(* CODESYS project RPI 3b stand it.project

Project tree, tasks and I/O mapping:
  Device : CODESYS Control for Raspberry Pi SL, 3S - Smart Software Solutions GmbH, version 3.5.12.30
    application Application
      libraries: Standard, * (System); VisuDialogs, * (System)
      task MainTask (cyclic, interval 4 ms, priority 1) calls PLC_PRG
      task TrendRecordingTask (cyclic, interval 100 ms, priority 0) calls VisuTrendStorageAccess.GlobalInstances.g_TrendRecordingManager.CyclicCall
      task VISU_TASK (cyclic, interval 50 ms, priority 0) calls VisuElems.Visu_Prg
      global variables GVL
      visualisation Operator_panel
      Trend Recording Manager
        Visualization_Trend3
        Visualization_Trend2
        Operator_panel_Trend3
      Symbols
      program PLC_PRG [FBD]
      visualisation Experiment_settings
      visualisation Login
      function AfterLogin [ST]
      visualisation Settings_WGR
      visualisation Visualization
      visualisation Well_not_killed_10min
      program MySQL [ST]
      program MySQL_VISU [CFC]
      visualisation MySQL_visu
    SPI
    I²C
    SoftMotion General Axis Pool
    Modbus_COM_1 : Modbus COM, 3S - Smart Software Solutions GmbH, version 3.5.11.20
        settings: DataBits = 8; StopBits = 1; ComPort = 1
      Modbus_Master_COM_Port : Modbus Master, COM Port, 3S - Smart Software Solutions GmbH, version 3.5.12.0
          settings: Transmission = 'RTU'; ResponseTimeout = 1000; TimeBetweenFrames = 10; Auto-restart communication = TRUE
        SI30_Water_In_Add4 : Modbus Slave, COM Port, 3S - Smart Software Solutions GmbH, version 3.5.10.30
            settings: SlaveAddress = 4; ResponseTimeout = 1000; UseExtendedFunctionCodes = TRUE; Channel 2.Function Code = 5; Channel 2.Read Offset = 0; Channel 2.Read Length = 0; Channel 2.Write Offset = 16#0002; Channel 2.Write Length = 1; Channel 2.Cycle Time = 100; Channel 1.Function Code = 4; Channel 1.Read Offset = 16#0000; Channel 1.Read Length = 2; Channel 1.Write Offset = 0; Channel 1.Write Length = 0; Channel 1.Cycle Time = 100
            output Application.PLC_PRG.Reset_SI30_Waterflow_in : ARRAY[0..0] OF BYTE  // Channel 2
            input  Application.PLC_PRG.MB_Counter1_water_in : WORD  // Channel 1.Channel 1
            input  Application.PLC_PRG.MB_Counter2_water_in : WORD  // Channel 1.Channel 1
            unmapped channels: Channel 1
        VA520_Add5 : Modbus Slave, COM Port, 3S - Smart Software Solutions GmbH, version 3.5.10.30
            settings: SlaveAddress = 5; ResponseTimeout = 1000; UseExtendedFunctionCodes = TRUE; Channel 0.Function Code = 3; Channel 0.Read Offset = 16#044B; Channel 0.Read Length = 2; Channel 0.Write Offset = 0; Channel 0.Write Length = 0; Channel 0.Cycle Time = 100; Channel 1.Function Code = 3; Channel 1.Read Offset = 16#0541; Channel 1.Read Length = 2; Channel 1.Write Offset = 0; Channel 1.Write Length = 0; Channel 1.Cycle Time = 100; Channel 2.Function Code = 3; Channel 2.Read Offset = 16#0589; Channel 2.Read Length = 2; Channel 2.Write Offset = 0; Channel 2.Write Length = 0; Channel 2.Cycle Time = 100; Channel 3.Function Code = 3; Channel 3.Read Offset = 16#04F5; Channel 3.Read Length = 2; Channel 3.Write Offset = 0; Channel 3.Write Length = 0; Channel 3.Cycle Time = 100; Channel 6.Function Code = 3; Channel 6.Read Offset = 16#03EA; Channel 6.Read Length = 2; Channel 6.Write Offset = 0; Channel 6.Write Length = 0; Channel 6.Cycle Time = 100
            input  Application.PLC_PRG.MB_input_Airflow : ARRAY[0..1] OF WORD  // Channel 0
            input  Application.PLC_PRG.MB_input_Velocity : ARRAY[0..1] OF WORD  // Channel 1
            input  Application.PLC_PRG.MB_input_Airtemp : ARRAY[0..1] OF WORD  // Channel 2
            input  Application.PLC_PRG.MB_input_Airconsumption_ac : ARRAY[0..1] OF WORD  // Channel 3
            input  Application.PLC_PRG.MB_input_Airconsumption2_bc : WORD  // Channel 6.Channel 6
            unmapped channels: Channel 6
        WP8028ADAM_Add2 : Modbus Slave, COM Port, 3S - Smart Software Solutions GmbH, version 3.5.10.30
            settings: SlaveAddress = 2; ResponseTimeout = 1000; UseExtendedFunctionCodes = TRUE; Channel 0.Function Code = 5; Channel 0.Read Offset = 0; Channel 0.Read Length = 0; Channel 0.Write Offset = 16#0000; Channel 0.Write Length = 1; Channel 0.Cycle Time = 100; Channel 1.Function Code = 5; Channel 1.Read Offset = 0; Channel 1.Read Length = 0; Channel 1.Write Offset = 16#0001; Channel 1.Write Length = 1; Channel 1.Cycle Time = 100; Channel 2.Function Code = 5; Channel 2.Read Offset = 0; Channel 2.Read Length = 0; Channel 2.Write Offset = 16#0002; Channel 2.Write Length = 1; Channel 2.Cycle Time = 100; Channel 3.Function Code = 5; Channel 3.Read Offset = 0; Channel 3.Read Length = 0; Channel 3.Write Offset = 16#0003; Channel 3.Write Length = 1; Channel 3.Cycle Time = 100; Channel 4.Function Code = 5; Channel 4.Read Offset = 0; Channel 4.Read Length = 0; Channel 4.Write Offset = 16#0004; Channel 4.Write Length = 1; Channel 4.Cycle Time = 100; Channel 5.Function Code = 5; Channel 5.Read Offset = 0; Channel 5.Read Length = 0; Channel 5.Write Offset = 16#0005; Channel 5.Write Length = 1; Channel 5.Cycle Time = 100; Channel 6.Function Code = 5;
              Channel 6.Read Offset = 0; Channel 6.Read Length = 0; Channel 6.Write Offset = 16#0006; Channel 6.Write Length = 1; Channel 6.Cycle Time = 100; Channel 7.Function Code = 2; Channel 7.Read Offset = 16#0000; Channel 7.Read Length = 1; Channel 7.Write Offset = 0; Channel 7.Write Length = 0; Channel 7.Cycle Time = 100; Channel 8.Function Code = 2; Channel 8.Read Offset = 16#0001; Channel 8.Read Length = 1; Channel 8.Write Offset = 0; Channel 8.Write Length = 0; Channel 8.Cycle Time = 100; Channel 9.Function Code = 5; Channel 9.Read Offset = 0; Channel 9.Read Length = 0; Channel 9.Write Offset = 16#0007; Channel 9.Write Length = 1; Channel 9.Cycle Time = 100
            output Application.PLC_PRG.SV1_Switch_onoff : ARRAY[0..0] OF BYTE  // Channel 0
            output Application.PLC_PRG.SV2_Switch_onoff : ARRAY[0..0] OF BYTE  // Channel 1
            output Application.PLC_PRG.SV3_Switch_onoff : ARRAY[0..0] OF BYTE  // Channel 2
            output Application.PLC_PRG.SV4_Switch_onoff : ARRAY[0..0] OF BYTE  // Channel 3
            output Application.PLC_PRG.SV5_Switch_onoff : ARRAY[0..0] OF BYTE  // Channel 4
            output Application.PLC_PRG.SV6_Switch_onoff : ARRAY[0..0] OF BYTE  // Channel 5
            output Application.PLC_PRG.SV7_Switch_onoff : ARRAY[0..0] OF BYTE  // Channel 6
            input  Application.PLC_PRG.Intercooler_heat_switch_DI01 : ARRAY[0..0] OF BYTE  // Channel 7
            input  Application.PLC_PRG.Intercooler_level_sensor_DI02 : ARRAY[0..0] OF BYTE  // Channel 8
            output Application.PLC_PRG.Intercooler_water_for_cooling_DO08 : ARRAY[0..0] OF BYTE  // Channel 9
        WP3082ADAM_Add3 : Modbus Slave, COM Port, 3S - Smart Software Solutions GmbH, version 3.5.10.30
            settings: SlaveAddress = 3; ResponseTimeout = 1000; UseExtendedFunctionCodes = TRUE; Channel 1.Function Code = 3; Channel 1.Read Offset = 16#0001; Channel 1.Read Length = 2; Channel 1.Write Offset = 0; Channel 1.Write Length = 0; Channel 1.Cycle Time = 100; Channel 2.Function Code = 3; Channel 2.Read Offset = 16#0002; Channel 2.Read Length = 2; Channel 2.Write Offset = 0; Channel 2.Write Length = 0; Channel 2.Cycle Time = 100; Channel 3.Function Code = 3; Channel 3.Read Offset = 16#0003; Channel 3.Read Length = 2; Channel 3.Write Offset = 0; Channel 3.Write Length = 0; Channel 3.Cycle Time = 100; Channel 4.Function Code = 3; Channel 4.Read Offset = 16#0004; Channel 4.Read Length = 2; Channel 4.Write Offset = 0; Channel 4.Write Length = 0; Channel 4.Cycle Time = 100; Channel 5.Function Code = 3; Channel 5.Read Offset = 16#0005; Channel 5.Read Length = 2; Channel 5.Write Offset = 0; Channel 5.Write Length = 0; Channel 5.Cycle Time = 100; Channel 6.Function Code = 3; Channel 6.Read Offset = 16#0006; Channel 6.Read Length = 2; Channel 6.Write Offset = 0; Channel 6.Write Length = 0; Channel 6.Cycle Time = 100
            input  Application.PLC_PRG.Analog_input_Ch01 : WORD  // Channel 1.Channel 1
            input  Application.PLC_PRG.Analog_input_Ch02 : WORD  // Channel 2.Channel 2
            input  Application.PLC_PRG.Analog_input_Ch03 : WORD  // Channel 3.Channel 3
            input  Application.PLC_PRG.Analog_input_Ch04 : WORD  // Channel 4.Channel 4
            input  Application.PLC_PRG.Analog_input_Ch05 : WORD  // Channel 5.Channel 5
            input  Application.PLC_PRG.Analog_input_Ch06 : WORD  // Channel 6.Channel 6
            unmapped channels: %IW2 Channel 1, %IW4 Channel 2, %IW6 Channel 3, %IW8 Channel 4, %IW10 Channel 5, %IW42 Channel 6
        HU4AO_Add1 : Modbus Slave, COM Port, 3S - Smart Software Solutions GmbH, version 3.5.10.30
            settings: 16#0007 (=7).Function Code = 6; 16#0007 (=7).Write Offset = 7; 16#0007 (=7).Write Length = 1; 16#0007 (=7).Init Value = 5; Channel 0.Function Code = 6; Channel 0.Read Offset = 0; Channel 0.Read Length = 0; Channel 0.Write Offset = 16#000F; Channel 0.Write Length = 1; Channel 0.Cycle Time = 100; Channel 1.Function Code = 3; Channel 1.Read Offset = 16#0010; Channel 1.Read Length = 2; Channel 1.Write Offset = 0; Channel 1.Write Length = 0; Channel 1.Cycle Time = 100
            output Application.PLC_PRG.Pump_speed_reference : ARRAY[0..0] OF WORD  // Channel 0
            unmapped channels: Channel 1
        SI30_Foam_In_Add6 : Modbus Slave, COM Port, 3S - Smart Software Solutions GmbH, version 3.5.10.30
            settings: SlaveAddress = 6; ResponseTimeout = 1000; UseExtendedFunctionCodes = TRUE; Channel 0.Function Code = 4; Channel 0.Read Offset = 16#0000; Channel 0.Read Length = 2; Channel 0.Write Offset = 0; Channel 0.Write Length = 0; Channel 0.Cycle Time = 100; Channel 1.Function Code = 5; Channel 1.Read Offset = 0; Channel 1.Read Length = 0; Channel 1.Write Offset = 16#0002; Channel 1.Write Length = 1; Channel 1.Cycle Time = 100
            input  Application.PLC_PRG.MB_Counter1_foam_in : WORD  // Channel 0.Channel 0
            input  Application.PLC_PRG.MB_Counter2_foam_in : WORD  // Channel 0.Channel 0
            output Application.PLC_PRG.Reset_SI30_Foam_in : ARRAY[0..0] OF BYTE  // Channel 1
            unmapped channels: Channel 0
        SI30_Water_Out_Add8 : Modbus Slave, COM Port, 3S - Smart Software Solutions GmbH, version 3.5.10.30
            settings: SlaveAddress = 8; ResponseTimeout = 1000; UseExtendedFunctionCodes = TRUE; Channel 0.Function Code = 4; Channel 0.Read Offset = 16#0000; Channel 0.Read Length = 2; Channel 0.Write Offset = 0; Channel 0.Write Length = 0; Channel 0.Cycle Time = 100; Channel 1.Function Code = 5; Channel 1.Read Offset = 0; Channel 1.Read Length = 0; Channel 1.Write Offset = 16#0002; Channel 1.Write Length = 1; Channel 1.Cycle Time = 100
            input  Application.PLC_PRG.MB_Counter1_water_out : WORD  // Channel 0.Channel 0
            input  Application.PLC_PRG.MB_Counter2_water_out : WORD  // Channel 0.Channel 0
            output Application.PLC_PRG.Reset_SI30_Waterflow_out : ARRAY[0..0] OF BYTE  // Channel 1
            unmapped channels: Channel 0
        SI30_Foam_Extinguisher_Add7 : Modbus Slave, COM Port, 3S - Smart Software Solutions GmbH, version 3.5.10.30
            settings: SlaveAddress = 7; ResponseTimeout = 1000; UseExtendedFunctionCodes = TRUE; Channel 0.Function Code = 4; Channel 0.Read Offset = 16#0000; Channel 0.Read Length = 2; Channel 0.Write Offset = 0; Channel 0.Write Length = 0; Channel 0.Cycle Time = 100; Channel 1.Function Code = 5; Channel 1.Read Offset = 0; Channel 1.Read Length = 0; Channel 1.Write Offset = 16#0002; Channel 1.Write Length = 1; Channel 1.Cycle Time = 100
            input  Application.PLC_PRG.MB_Counter1_foam_exting : WORD  // Channel 0.Channel 0
            input  Application.PLC_PRG.MB_Counter2_foam_exting : WORD  // Channel 0.Channel 0
            output Application.PLC_PRG.Reset_SI30_Foam_extinguisher : ARRAY[0..0] OF BYTE  // Channel 1
            unmapped channels: Channel 0
        WP8028ADAM_Add10 : Modbus Slave, COM Port, 3S - Smart Software Solutions GmbH, version 3.5.10.30
            settings: SlaveAddress = 10; ResponseTimeout = 1000; UseExtendedFunctionCodes = TRUE; Channel 0.Function Code = 5; Channel 0.Read Offset = 0; Channel 0.Read Length = 0; Channel 0.Write Offset = 16#0000; Channel 0.Write Length = 1; Channel 0.Cycle Time = 100; Channel 1.Function Code = 5; Channel 1.Read Offset = 0; Channel 1.Read Length = 0; Channel 1.Write Offset = 16#0001; Channel 1.Write Length = 1; Channel 1.Cycle Time = 100; Channel 2.Function Code = 5; Channel 2.Read Offset = 0; Channel 2.Read Length = 0; Channel 2.Write Offset = 16#0002; Channel 2.Write Length = 1; Channel 2.Cycle Time = 100; Channel 3.Function Code = 5; Channel 3.Read Offset = 0; Channel 3.Read Length = 0; Channel 3.Write Offset = 16#0003; Channel 3.Write Length = 1; Channel 3.Cycle Time = 100; Channel 4.Function Code = 5; Channel 4.Read Offset = 0; Channel 4.Read Length = 0; Channel 4.Write Offset = 16#0004; Channel 4.Write Length = 1; Channel 4.Cycle Time = 100; Channel 5.Function Code = 5; Channel 5.Read Offset = 0; Channel 5.Read Length = 0; Channel 5.Write Offset = 16#0005; Channel 5.Write Length = 1; Channel 5.Cycle Time = 100; Channel 6.Function Code = 5;
              Channel 6.Read Offset = 0; Channel 6.Read Length = 0; Channel 6.Write Offset = 16#0006; Channel 6.Write Length = 1; Channel 6.Cycle Time = 100; Channel 7.Function Code = 5; Channel 7.Read Offset = 0; Channel 7.Read Length = 0; Channel 7.Write Offset = 16#0007; Channel 7.Write Length = 1; Channel 7.Cycle Time = 100
            output Application.PLC_PRG.Switch_ONOFF_Compressor : ARRAY[0..0] OF BYTE  // Channel 2
            output Application.PLC_PRG.Switch_ONOFF_Intercooler_Heater : ARRAY[0..0] OF BYTE  // Channel 3
            unmapped channels: Channel 0, Channel 1, Channel 4, Channel 5, Channel 6, Channel 7
        WP3082ADAM_Add9 : Modbus Slave, COM Port, 3S - Smart Software Solutions GmbH, version 3.5.10.30
            settings: SlaveAddress = 9; ResponseTimeout = 1000; UseExtendedFunctionCodes = TRUE; Channel 0.Function Code = 3; Channel 0.Read Offset = 16#0000; Channel 0.Read Length = 2; Channel 0.Write Offset = 0; Channel 0.Write Length = 0; Channel 0.Cycle Time = 100; Channel 1.Function Code = 3; Channel 1.Read Offset = 16#0001; Channel 1.Read Length = 2; Channel 1.Write Offset = 0; Channel 1.Write Length = 0; Channel 1.Cycle Time = 100; Channel 2.Function Code = 3; Channel 2.Read Offset = 16#0002; Channel 2.Read Length = 2; Channel 2.Write Offset = 0; Channel 2.Write Length = 0; Channel 2.Cycle Time = 100; Channel 3.Function Code = 3; Channel 3.Read Offset = 16#0003; Channel 3.Read Length = 2; Channel 3.Write Offset = 0; Channel 3.Write Length = 0; Channel 3.Cycle Time = 100; Channel 4.Function Code = 3; Channel 4.Read Offset = 16#0004; Channel 4.Read Length = 2; Channel 4.Write Offset = 0; Channel 4.Write Length = 0; Channel 4.Cycle Time = 100; Channel 5.Function Code = 3; Channel 5.Read Offset = 16#0005; Channel 5.Read Length = 2; Channel 5.Write Offset = 0; Channel 5.Write Length = 0; Channel 5.Cycle Time = 100; Channel 6.Function Code = 3;
              Channel 6.Read Offset = 16#0006; Channel 6.Read Length = 2; Channel 6.Write Offset = 0; Channel 6.Write Length = 0; Channel 6.Cycle Time = 100
            unmapped channels: Channel 0, Channel 1, Channel 2, Channel 3, Channel 4, Channel 5, Channel 6
    Onewire
    GPIOs_A_B : GPIOs A/B, 3S - Smart Software Solutions GmbH, version 3.5.11.0
        unmapped channels: digital inputs (GPIO0..GPIO31), digital outputs (GPIO0..GPIO31)
    Camera device
      <Empty>
  libraries: VisuSymbols, 3.5.10.0 (System); BASIC, 3.31 (OSCAT); S4A_SQL4CodesysV3, 4.0.0.1 (SQL4automation); MySQL Library, 1.1.0.0 (Pfänder GmbH)
  text list GlobalTextList
  image pool ImagePool
  AC_GENERATOR_DATA
  5ce3da45-db07-42e7-a21c-a00fff4ed8f6|C:\Program Files\3S CODESYS\CODESYS\Visu\Pictures\Visualization.jpg
  5ce3da45-db07-42e7-a21c-a00fff4ed8f6|C:\Program Files\3S CODESYS\CODESYS\Visu\Pictures\Wellhead.jpg
  5ce3da45-db07-42e7-a21c-a00fff4ed8f6|C:\Program Files\3S CODESYS\CODESYS\Visu\Pictures\GWS.jpg
*)

// Device/Application/GVL
{attribute 'qualified_only'}
VAR_GLOBAL
	Well_temperature: REAL;
	Mast_temperature: REAL;
END_VAR

// Device/Application/PLC_PRG
PROGRAM PLC_PRG

VAR
	// Speed reference 0-10V
	Pump_speed_reference: WORD := 0;
	Analog_input_Ch01: WORD := 0;
	// Celsium Centigrates
	Mast_temperature: REAL := 0;
	Analog_input_Ch02: WORD := 0;
	// Celsium Centigrates
	Well_temperature: REAL := 0;
	Analog_input_Ch03: WORD := 0;
	// KPa
	Separator_pressure: REAL := 0;
	Analog_input_Ch04: WORD := 0;
	// KPa
	Receiver_pressure: REAL := 0;
	Analog_input_Ch05: WORD := 0;
	// KPa
	Differential_pressure: REAL := 0;
	// counts
	MB_Counter1_water_in: WORD := 0;
	// counts
	MB_Counter2_water_in: WORD := 0;
	// Volume from water counter
	Water_in_volume_counts: REAL := 0;
	// Volume from foam counter
	Foam_volume_counts: Real := 0;
	// Open/Close solenoid valve for air flow to separator
	SV4_Switch_onoff: BOOL := 0;
	// Open/Close solenoid valve for foam extinguishing in separators
	SV3_Switch_onoff: BOOL := 0;
	// Open/Close solenoid valve for water flow to well
	SV2_Switch_onoff: BOOL := 0;
	// Open/Close solenoid valve for foam flow to well
	SV1_Switch_onoff: BOOL := 0;
	// Open/Close solenoid valve for air flow to receiver
	SV5_Switch_onoff: BOOL := 0;
	// Open/Close solenoid valve for drain air from separator
	SV6_Switch_onoff: BOOL := 0;
	// Open/Close solenoid valve for drain air from receiver
	SV7_Switch_onoff: BOOL := 0;
	MB_input_Airflow: DWORD := 0;
	MB_input_Velocity: DWORD := 0;
	MB_input_Airtemp: DWORD := 0;
	// From flowmeter
	Air_flow: REAL := 0;
	// From flowmeter
	Air_velocity: REAL := 0;
	// From flowmeter
	Air_temp: REAL := 0;
	PID_regulator: CTRL_PID;
	// Pressure @ system given by Operator
	OP_System_Pressure: Real := 0;
	// Temperature of air given by Operator
	OP_System_Temperature: Real := 0;
	// Airflow via Flowmeter given by Operator
	OP_System_Airflow: Real := 0;
	// Waterflow via counter given by Operator
	OP_System_Waterflow: Real := 0;
	// Foamflow via counter given by Operator
	OP_System_Foamflow: Real := 0;
	// Water gas ratio set by Operator
	OP_WGR_Setpoint: Real := 0;
	// Actual water gas ratio cm3/m3
	WGR_Actual: Real := 0;
	// Pump reference setpoint given by Operator
	OP_Speed_Pump: Real := 0;
	// Start experiment
	START: Bool := 0;
	// Stop experiment
	STOP: Bool := 0;
	// Reset all values to zero
	RESET_to_zero: BOOL := 0;
	SR_0: SR;
	// Shutdown when one of alarms become active
	Common_Alarm_Shutdown: Bool := 0;
	Fixed_0: Bool := 0;
	Fixed_1: Bool := 1;
	// Stricted system pressure
	System_pressure: Real := 0;
	TON_0: TON;
	CTRL_PWM_0: CTRL_PWM;
	Pulse: BOOL := 0;
	// Variable for calculating actual Waterflow
	Waterflow_calc_actual: Real := 0;
	Pa_Time_calc_actual_Waterflow: time := t#1s;
	// Pulse generator for counting waterflow
	GP_0: gen_pulse;
	// Total waterflow in cm3 from counter
	Waterflow_in: real := 0;
	// Pulse generator for making tacts to SV2 (water sprying to well)
	GP_1: Gen_pulse;
	SR_1: SR;
	SR_2: SR;
	// SR trigger for counting time of experiment
	SR_3: SR;
	// Counting time of the experiment 10 min
	TON_1: TON;
	Exp_time_elapsed_10min: bool := 0;
	// Counting time of the experiment 60 min
	TON_2: TON;
	Exp_time_elapsed_60min: bool := 0;
	SR_4: SR;
	SR_5: SR;
	Well_killed: bool := 0;
	TON_3: TON;
	// Reset of the water flowmeter counter
	Reset_SI30_Waterflow_in: BOOL := 0;
	RS_0: RS;
	RS_1: RS;
	RS_2: RS;
	RS_3: RS;
	RS_4: RS;
	RS_5: RS;
	Reset_SI30_Foam_in: BOOL;
	// Total consumption of air from flowmeter in m3 after comma
	MB_input_Airconsumption_ac: DWORD := 0;
	// From flowmeter consumption after comma
	Air_consumption_ac: REAL := 0;
	// Total consumption of air from flowmeter in m3 before comma
	MB_input_Airconsumption1_bc: WORD := 0;
	// Total consumption of air from flowmeter in m3 before comma
	MB_input_Airconsumption2_bc: WORD := 0;
	// From flowmeter consumption before comma
	Air_consumption_bc: REAL := 0;
	R_TRIG_0: R_TRIG;
	// From this value starts counting air consumption
	Air_consumption_startpoint: REAL;
	// Calculated air consumption in m3
	Air_consumption_calc: REAL;
	// Counts water from separator
	MB_Counter1_water_out: WORD;
	// Counts water from separator
	MB_Counter2_water_out: WORD;
	Water_out_volume_counts: REAL;
	// Reset of the waterflow meter counter
	Reset_SI30_Waterflow_out: BOOL := 0;
	// Total water volume in system
	Water_volume_in_system: REAL;
	TON_4: TON;
	TON_5: TON;
	TON_6: TON;
	R_TRIG_1: R_TRIG;
	Air_flow_startpoint: REAL;
	RS_6: RS;
	TOF_0: TOF;
	// System pressure is reached value set by Operator
	Pressure_ready: BOOL;
	RS_7: RS;
	RS_8: RS;
	TOF_1: TOF;
	// Type of experiment chosen by Operator
	Type_of_exp: INT;
	RS_9: RS;
	// Release pressure from system
	Release_pressure: BOOL;
	RS_10: RS;
	// Push foam into well
	Push_foam: BOOL;
	TON_7: TON;
	TOF_2: TOF;
	RS_11: RS;
	// Intercooler temperature, Celsium Centigrates
	Analog_input_Ch06: WORD := 0;
	// Celsium Centigrates
	Intercoller_temperature: REAL := 0;
	// Switch on/off intercooler heater
	Switch_ONOFF_Intercooler_Heater: BOOL := 0;
	// Counts from foam counter
	MB_Counter1_foam_in: WORD := 0;
	// Counts from foam counter
	MB_Counter2_foam_in: WORD := 0;
	// Counts from foam extinguisher counter
	MB_Counter1_foam_exting: WORD := 0;
	// Counts from foam extinguisher counter
	MB_Counter2_foam_exting: WORD := 0;
	Reset_SI30_Foam_extinguisher: BOOL := 0;
	Switch_ONOFF_Compressor: BOOL := 0;
	Water_to_extinguish_foam_counts: REAL := 0;
	// From flowmeter VA520
	Air_consumption: REAL := 0;
	// Reset alarms and failures
	Common_RESET: BOOL := 0;
	// Intercooler heat switch ONOFF
	Intercooler_heat_switch_DI01: BOOL := 0;
	// Intercooler level sensor ONOFF
	Intercooler_level_sensor_DI02: BOOL := 0;
	// Solenoid opens water to cool down Intercooler
	Intercooler_water_for_cooling_DO08: BOOL := 0;
	RS_12: RS;
	RS_13: RS;
	RS_14: RS;
END_VAR
VAR // added by the converter: edge detectors and wires of the graphical bodies
    _w1, _w2, _w3 : INT;
END_VAR

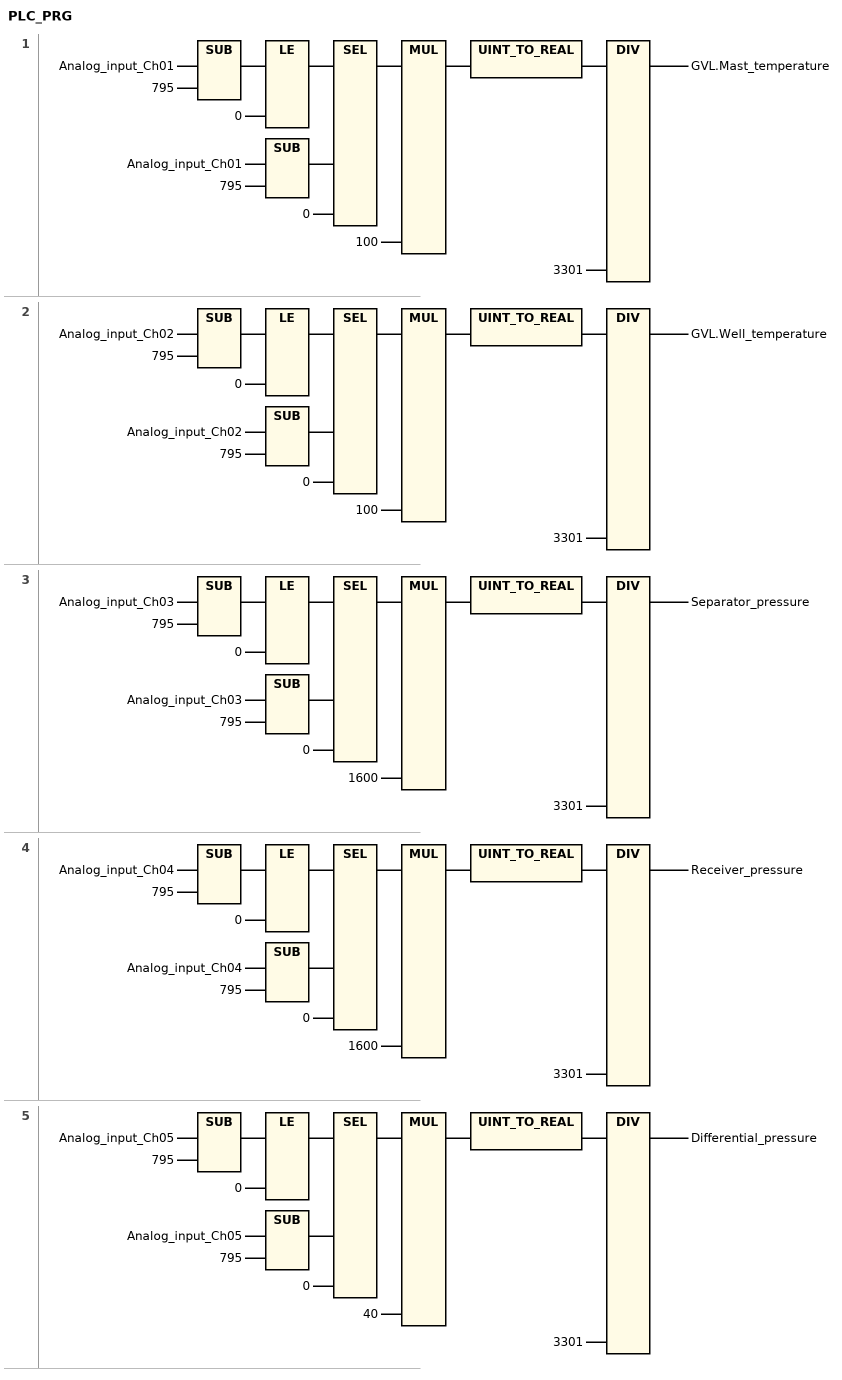
// NETWORK 1
GVL.Mast_temperature := UINT_TO_REAL(SEL(Analog_input_Ch01 - 795 <= 0, Analog_input_Ch01 - 795, 0) * 100) / 3301;

// NETWORK 2
GVL.Well_temperature := UINT_TO_REAL(SEL(Analog_input_Ch02 - 795 <= 0, Analog_input_Ch02 - 795, 0) * 100) / 3301;

// NETWORK 3
Separator_pressure := UINT_TO_REAL(SEL(Analog_input_Ch03 - 795 <= 0, Analog_input_Ch03 - 795, 0) * 1600) / 3301;

// NETWORK 4
Receiver_pressure := UINT_TO_REAL(SEL(Analog_input_Ch04 - 795 <= 0, Analog_input_Ch04 - 795, 0) * 1600) / 3301;

// NETWORK 5
Differential_pressure := UINT_TO_REAL(SEL(Analog_input_Ch05 - 795 <= 0, Analog_input_Ch05 - 795, 0) * 40) / 3301;

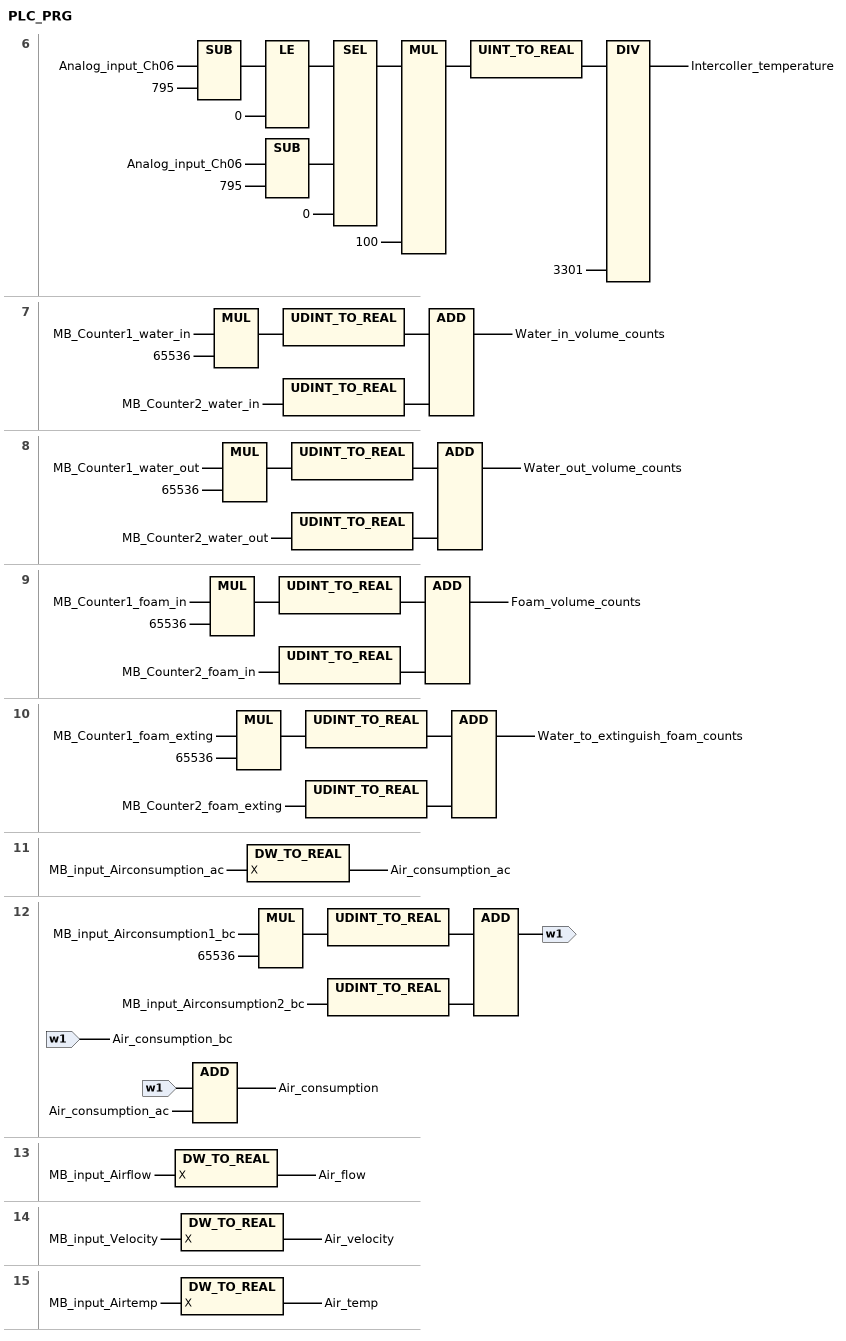
// NETWORK 6
Intercoller_temperature := UINT_TO_REAL(SEL(Analog_input_Ch06 - 795 <= 0, Analog_input_Ch06 - 795, 0) * 100) / 3301;

// NETWORK 7
Water_in_volume_counts := UDINT_TO_REAL(MB_Counter1_water_in * 65536) + UDINT_TO_REAL(MB_Counter2_water_in);

// NETWORK 8
Water_out_volume_counts := UDINT_TO_REAL(MB_Counter1_water_out * 65536) + UDINT_TO_REAL(MB_Counter2_water_out);

// NETWORK 9
Foam_volume_counts := UDINT_TO_REAL(MB_Counter1_foam_in * 65536) + UDINT_TO_REAL(MB_Counter2_foam_in);

// NETWORK 10
Water_to_extinguish_foam_counts := UDINT_TO_REAL(MB_Counter1_foam_exting * 65536) + UDINT_TO_REAL(MB_Counter2_foam_exting);

// NETWORK 11
Air_consumption_ac := DW_TO_REAL(X := MB_input_Airconsumption_ac);

// NETWORK 12
_w1 := UDINT_TO_REAL(MB_input_Airconsumption1_bc * 65536) + UDINT_TO_REAL(MB_input_Airconsumption2_bc);
Air_consumption_bc := _w1;
Air_consumption := _w1 + Air_consumption_ac;

// NETWORK 13
Air_flow := DW_TO_REAL(X := MB_input_Airflow);

// NETWORK 14
Air_velocity := DW_TO_REAL(X := MB_input_Velocity);

// NETWORK 15
Air_temp := DW_TO_REAL(X := MB_input_Airtemp);

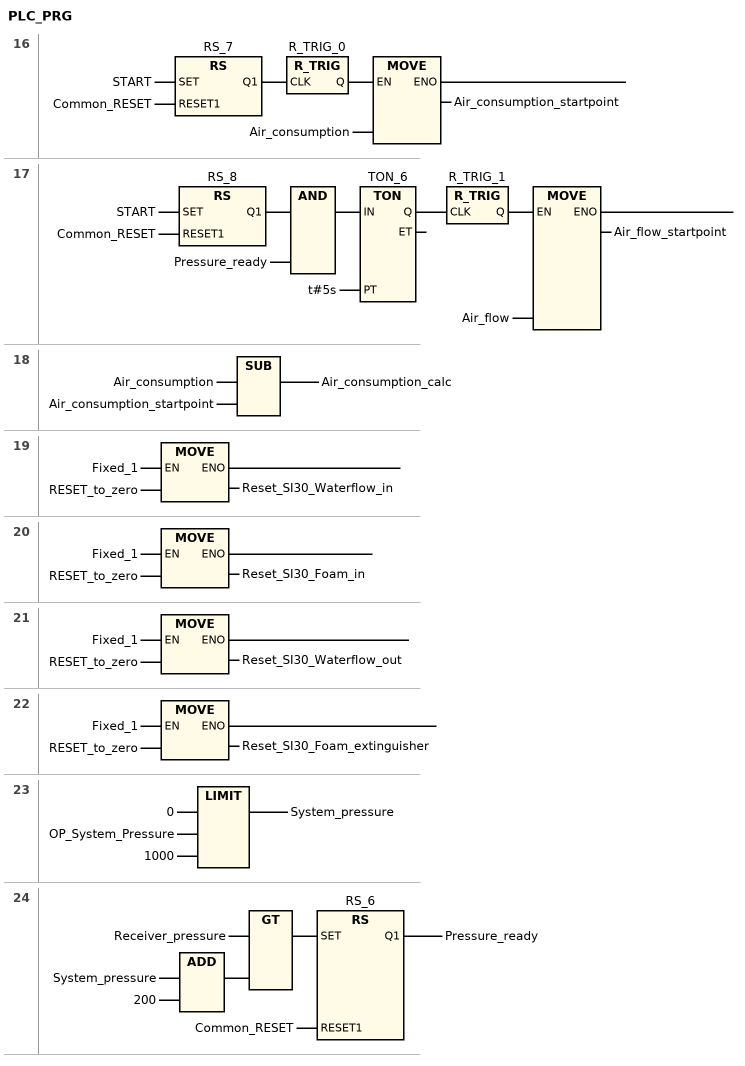
// NETWORK 16
RS_7(SET := START, RESET1 := Common_RESET); // RS
R_TRIG_0(CLK := RS_7.Q1); // R_TRIG
IF R_TRIG_0.Q THEN Air_consumption_startpoint := Air_consumption; END_IF

// NETWORK 17
RS_8(SET := START, RESET1 := Common_RESET); // RS
TON_6(IN := RS_8.Q1 AND Pressure_ready, PT := t#5s); // TON
R_TRIG_1(CLK := TON_6.Q); // R_TRIG
IF R_TRIG_1.Q THEN Air_flow_startpoint := Air_flow; END_IF

// NETWORK 18
Air_consumption_calc := Air_consumption - Air_consumption_startpoint;

// NETWORK 19
IF Fixed_1 THEN Reset_SI30_Waterflow_in := RESET_to_zero; END_IF

// NETWORK 20
IF Fixed_1 THEN Reset_SI30_Foam_in := RESET_to_zero; END_IF

// NETWORK 21
IF Fixed_1 THEN Reset_SI30_Waterflow_out := RESET_to_zero; END_IF

// NETWORK 22
IF Fixed_1 THEN Reset_SI30_Foam_extinguisher := RESET_to_zero; END_IF

// NETWORK 23
System_pressure := LIMIT(0, OP_System_Pressure, 1000);

// NETWORK 24
RS_6(SET := Receiver_pressure > System_pressure + 200, RESET1 := Common_RESET); // RS
Pressure_ready := RS_6.Q1;

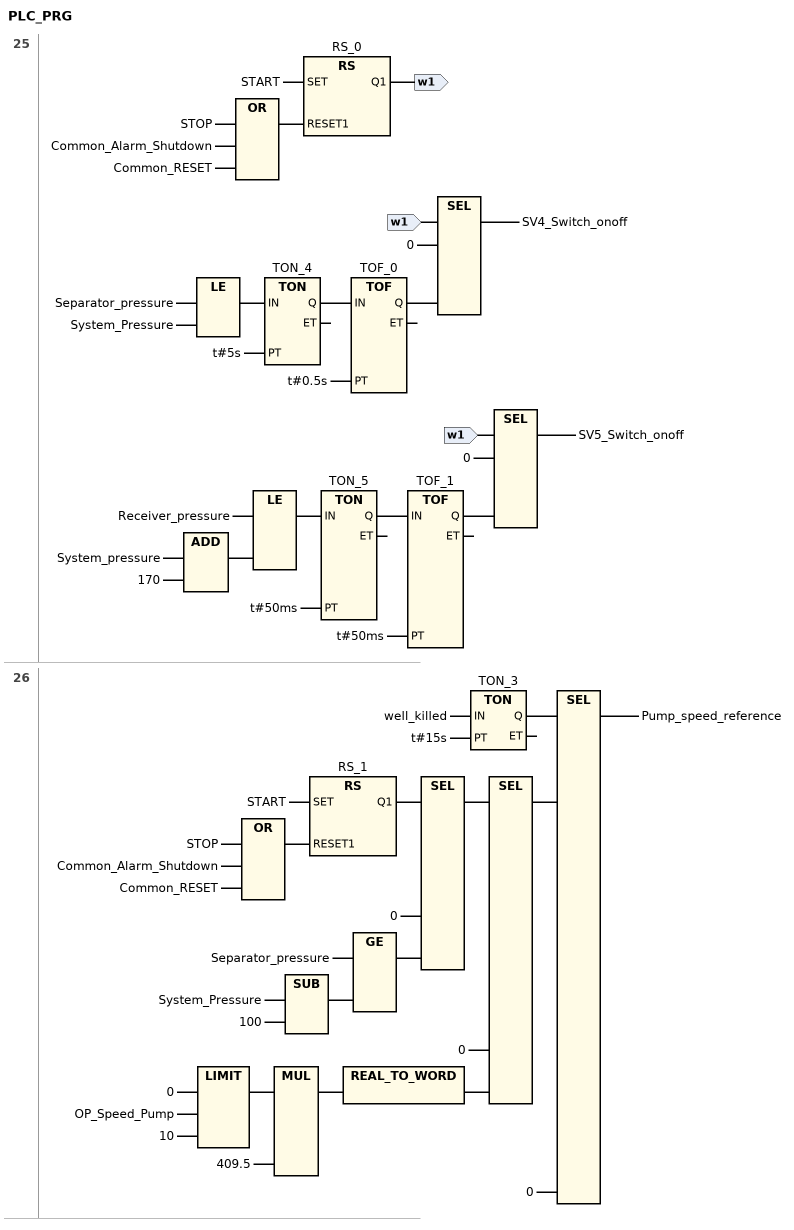
// NETWORK 25
RS_0(SET := START, RESET1 := STOP OR Common_Alarm_Shutdown OR Common_RESET); // RS
TON_4(IN := Separator_pressure <= System_Pressure, PT := t#5s); // TON
TOF_0(IN := TON_4.Q, PT := t#0.5s); // TOF
SV4_Switch_onoff := SEL(RS_0.Q1, 0, TOF_0.Q);
TON_5(IN := Receiver_pressure <= System_pressure + 170, PT := t#50ms); // TON
TOF_1(IN := TON_5.Q, PT := t#50ms); // TOF
SV5_Switch_onoff := SEL(RS_0.Q1, 0, TOF_1.Q);

// NETWORK 26
TON_3(IN := well_killed, PT := t#15s); // TON
RS_1(SET := START, RESET1 := STOP OR Common_Alarm_Shutdown OR Common_RESET); // RS
Pump_speed_reference := SEL(TON_3.Q, SEL(SEL(RS_1.Q1, 0, Separator_pressure >= System_Pressure - 100), 0, REAL_TO_WORD(LIMIT(0, OP_Speed_Pump, 10) * 409.5)), 0);

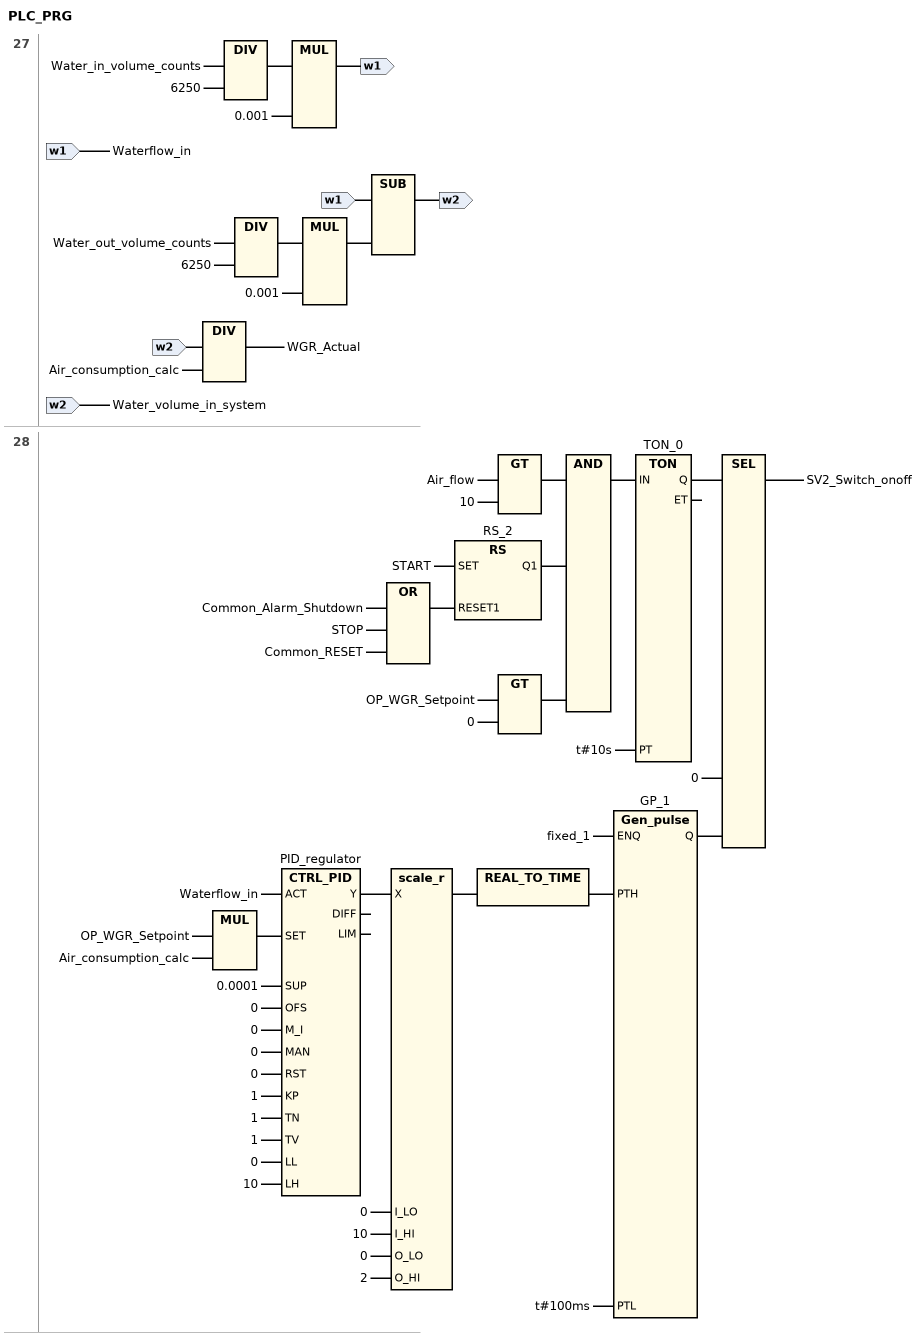
// NETWORK 27
_w2 := (Water_in_volume_counts / 6250) * 0.001;
Waterflow_in := _w2;
_w3 := _w2 - (Water_out_volume_counts / 6250) * 0.001;
WGR_Actual := _w3 / Air_consumption_calc;
Water_volume_in_system := _w3;

// NETWORK 28
RS_2(SET := START, RESET1 := Common_Alarm_Shutdown OR STOP OR Common_RESET); // RS
TON_0(IN := Air_flow > 10 AND RS_2.Q1 AND OP_WGR_Setpoint > 0, PT := t#10s); // TON
PID_regulator(
    ACT := Waterflow_in,
    SET := OP_WGR_Setpoint * Air_consumption_calc,
    SUP := 0.0001,
    OFS := 0,
    M_I := 0,
    MAN := 0,
    RST := 0,
    KP := 1,
    TN := 1,
    TV := 1,
    LL := 0,
    LH := 10); // CTRL_PID
GP_1(
    ENQ := fixed_1,
    PTH := REAL_TO_TIME(scale_r(X := PID_regulator.Y, I_LO := 0, I_HI := 10, O_LO := 0, O_HI := 2)),
    PTL := t#100ms); // Gen_pulse
SV2_Switch_onoff := SEL(TON_0.Q, 0, GP_1.Q);

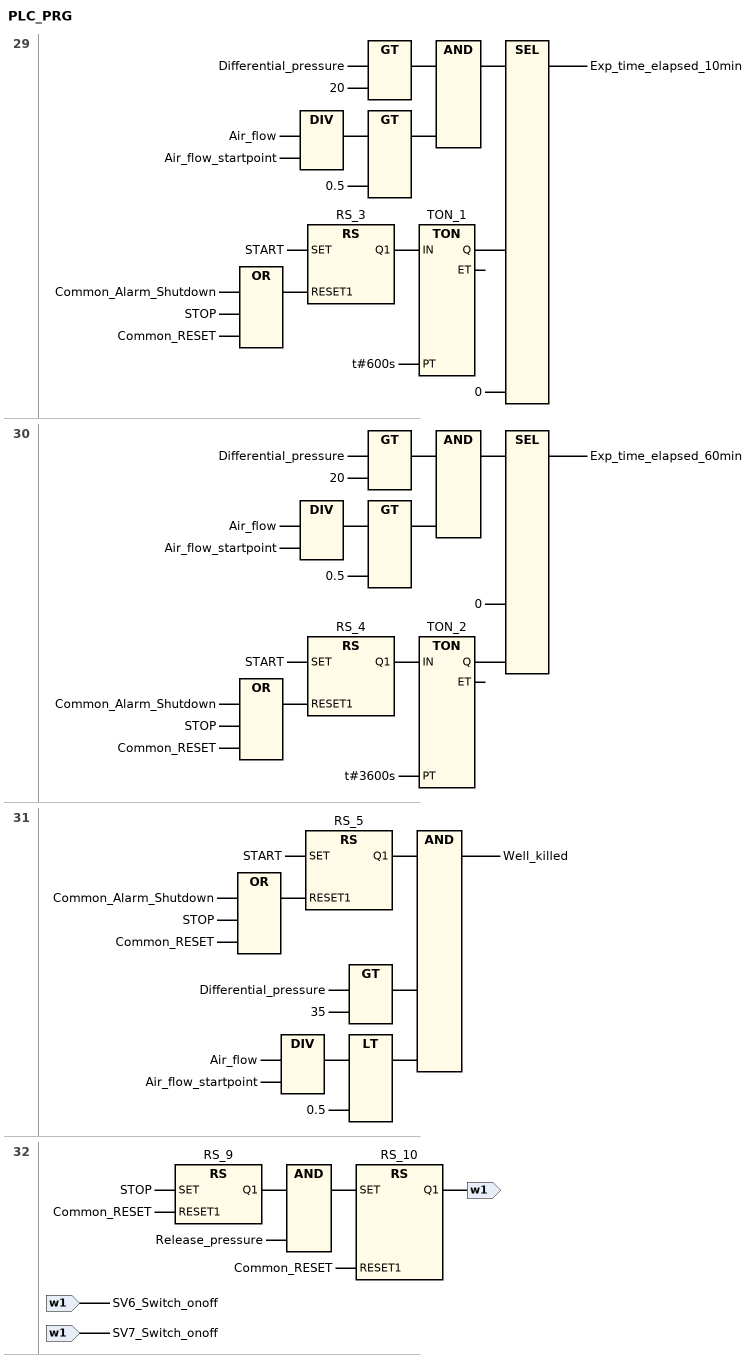
// NETWORK 29
RS_3(SET := START, RESET1 := Common_Alarm_Shutdown OR STOP OR Common_RESET); // RS
TON_1(IN := RS_3.Q1, PT := t#600s); // TON
Exp_time_elapsed_10min := SEL(Differential_pressure > 20 AND Air_flow / Air_flow_startpoint > 0.5, TON_1.Q, 0);

// NETWORK 30
RS_4(SET := START, RESET1 := Common_Alarm_Shutdown OR STOP OR Common_RESET); // RS
TON_2(IN := RS_4.Q1, PT := t#3600s); // TON
Exp_time_elapsed_60min := SEL(Differential_pressure > 20 AND Air_flow / Air_flow_startpoint > 0.5, 0, TON_2.Q);

// NETWORK 31
RS_5(SET := START, RESET1 := Common_Alarm_Shutdown OR STOP OR Common_RESET); // RS
Well_killed := RS_5.Q1 AND Differential_pressure > 35 AND Air_flow / Air_flow_startpoint < 0.5;

// NETWORK 32
RS_9(SET := STOP, RESET1 := Common_RESET); // RS
RS_10(SET := RS_9.Q1 AND Release_pressure, RESET1 := Common_RESET); // RS
SV6_Switch_onoff := RS_10.Q1;
SV7_Switch_onoff := RS_10.Q1;

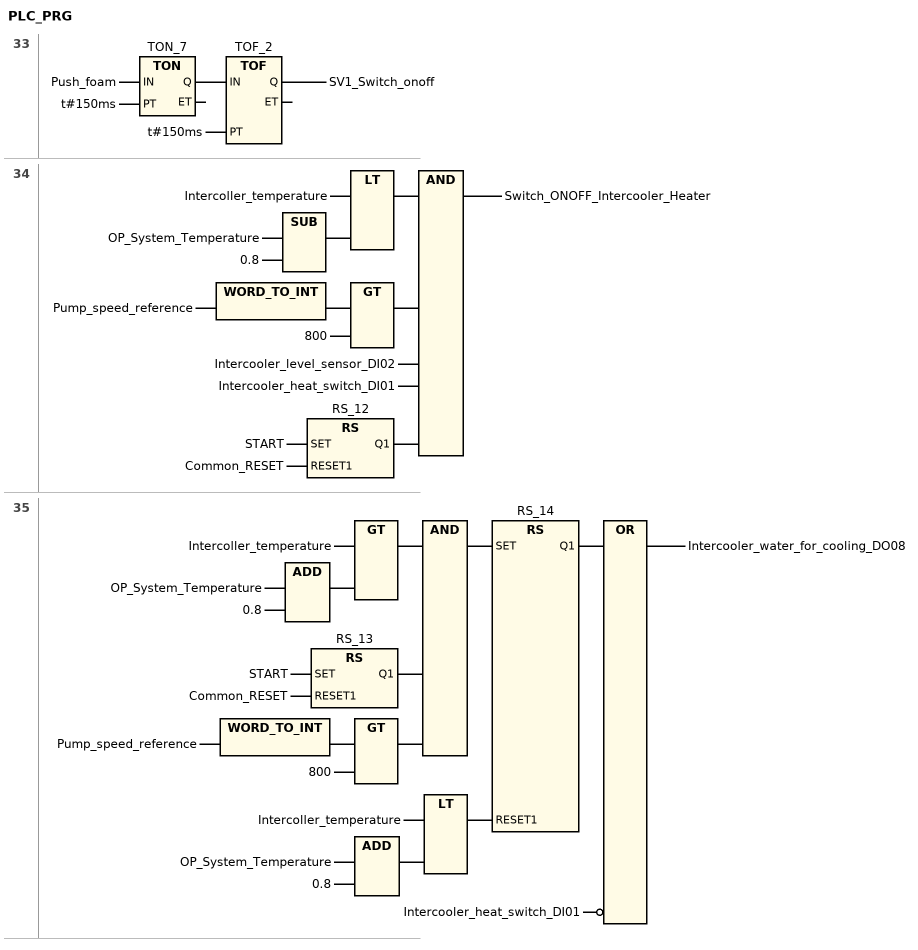
// NETWORK 33
TON_7(IN := Push_foam, PT := t#150ms); // TON
TOF_2(IN := TON_7.Q, PT := t#150ms); // TOF
SV1_Switch_onoff := TOF_2.Q;

// NETWORK 34
RS_12(SET := START, RESET1 := Common_RESET); // RS
Switch_ONOFF_Intercooler_Heater := Intercoller_temperature < OP_System_Temperature - 0.8 AND WORD_TO_INT(Pump_speed_reference) > 800 AND Intercooler_level_sensor_DI02 AND Intercooler_heat_switch_DI01 AND RS_12.Q1;

// NETWORK 35
RS_13(SET := START, RESET1 := Common_RESET); // RS
RS_14(SET := Intercoller_temperature > OP_System_Temperature + 0.8 AND RS_13.Q1 AND WORD_TO_INT(Pump_speed_reference) > 800, RESET1 := Intercoller_temperature < OP_System_Temperature + 0.8); // RS
Intercooler_water_for_cooling_DO08 := RS_14.Q1 OR NOT Intercooler_heat_switch_DI01;

END_PROGRAM

// Device/Application/AfterLogin
FUNCTION AfterLogin : BOOL
VAR_INPUT
	pClientData: POINTER TO VisuElems.VisuStructClientData;
END_VAR

IF VisuElems.CurrentUserGroupId <> 0 THEN
	VisuElems.g_VisuManager.SetMainVisu(pClientData, 'Operator_Panel');
END_IF

END_FUNCTION

// Device/Application/MySQL
PROGRAM MySQL
VAR
	
	// ** Instances
	MySQL_ConnString		: MySQL.MySQL_ConnectionString;		// MySQL_ConnString Handler FB - Do not edit it 
	MySQL_Open				: MySQL.MySQL_Open;					// MySQL_Open FB - Open the database connection
	MySQL_Close				: MySQL.MySQL_Close;				// MySQL_Close FB - Close the database connection
	MySQL_Exec				: MySQL.MySQL_Exec;					// MySQL_Exec FB - Execute a SQL-Command without no Result like (INSERT,UPDATE,DELETE,...)
	MySql_Query				: MySQL.MySql_Query;				// MySQL_Query FB - Execute a SQL-Command with DataSet Result like (SELECT,...) 
	
	// ** Connection Parameters
	_sHost					: STRING := 'localhost';			// Hostname or IP-adress
	_uiPort					: UINT 	 := 3306;					// MySQL Server Port
	_sDatabase				: STRING := 'testdb';				// Database Name
	_sUsername				: STRING := 'root';					// Database Username
	_sPassword				: STRING := 'root';					// User password 
	
	// ** Demo Project actions
	xDoOpen		 			: BOOL;								// TRUE = open the database connection	
	xDoClose 				: BOOL;								// TRUE = close the databasess connection
	xDoExecute	 			: BOOL;								// Starts the execute process on rising edge
	xDoQuery				: BOOL;								// Starts the query process on rising edge
	xDoExecuteWithTrigger	: BOOL;								// Starts the execute process with trigger - (CAUTION: Just for demo purpose, beacuse it executes as fast as possible)
	
	// ** States
	_xConnectionState		: BOOL;								// Shows the current database connection state as internal var
	_rtrigDoExecute			: R_TRIG;							// rtrig Execute 
	_xDoExecuteStateTrigger	: BOOL;								// Trigger State
	
	
	// ** MySQL_Commands Static	
	MySQL_Command_Query		: ARRAY [0..gc_MySQL_iStatementMax] OF STRING(gc_MySQL_iStatementLength) := ['SELECT * from data'];
	MySQL_Command_Exec		: ARRAY [0..gc_MySQL_iStatementMax] OF STRING(gc_MySQL_iStatementLength) := ['INSERT INTO data (Column_1, Column_2, Column_3) VALUES (1, 5, 10)'];
	MySQL_Command_Exec_Dyn	: ARRAY [0..gc_MySQL_iStatementMax] OF STRING(gc_MySQL_iStatementLength);

	iCounterVar1 			: INT;
	iCounterVar2 	 		: INT;		
	// ** MySQL_GetStringValue function parameters
	_iRow					: INT; 								// Row index
	_iColumn				: INT;								// Column index
	stResult 				: MySQL.MySQL_DataSet; 				// Result Structure
	ReadableString			: STRING(500); 						// Readable String	
END_VAR

// Open the Database connection on xDoOpen raising_edge
MySQL_Open(
	sHost:= _sHost, 
	uiPort:= _uiPort, 
	sDatabase:= _sDatabase, 
	sUsername:= _sUsername, 
	sPassword:= _sPassword, 
	xStart:= xDoOpen, 
	MySQL_Connection:= MySQL_ConnString, 
	xConnected=> _xConnectionState
);
	

// Example with static MySQL Command xDoExecute  	
IF NOT(xDoExecuteWithTrigger) AND _xConnectionState THEN
	 MySQL_Exec(
		xExecute:= xDoExecute, 
		MySQL_Connection:= MySQL_ConnString, 
		MySQL_Command:= MySQL_Command_Exec
	);			
END_IF

// Example with Trigger and dynamic MySQL command (IF xDoExecuteWithTrigger is active) - does Executes as fast as possible | Caution: This is stressing your database! 
IF _xConnectionState AND xDoExecuteWithTrigger THEN // Check if connection is open
	iCounterVar1 := iCounterVar1 +1;
	iCounterVar2 := iCounterVar2 +2;  
	
	MySQL_Command_Exec_Dyn[0] := 'INSERT INTO data (Column_1, Column_2, Column_3) VALUES (';
	MySQL_Command_Exec_Dyn[1] := '111,'; // --> Allways 111 
	MySQL_Command_Exec_Dyn[2] := CONCAT(INT_TO_STRING(iCounterVar1), ',');
	MySQL_Command_Exec_Dyn[3] := CONCAT(INT_TO_STRING(iCounterVar2), ')');
		
	IF MySQL_Exec.xDone OR MySQL_Exec.xError THEN
		_xDoExecuteStateTrigger := FALSE;
	ELSE
		IF MySQL_Exec.xExecute OR MySQL_Exec.xBusy THEN
			_xDoExecuteStateTrigger := FALSE;
		ELSE 
			_xDoExecuteStateTrigger := TRUE;
		END_IF
	END_IF
	_rtrigDoExecute(CLK:=_xDoExecuteStateTrigger);
 	MySQL_Exec(
		xExecute:= _rtrigDoExecute.Q, 
		MySQL_Connection:= MySQL_ConnString, 
		MySQL_Command:= MySQL_Command_Exec_Dyn,
	);			
END_IF

// Execute MySQL Command with Result
IF _xConnectionState THEN
	MySql_Query(
		xExecute:= xDoQuery, 
		MySQL_Command:= MySQL_Command_Query, 
		MySQL_Connection:= MySQL_ConnString, 
		stResultSet:= stResult
	);
	MySql_GetStringValue(_iRow,_iColumn, stResult, ReadableString);  
	
END_IF
	
// Close the MySQL-Connection
IF xDoClose AND _xConnectionState THEN
	MySQL_Close(
		xStart:= xDoClose, 
		MySQL_Connection:= MySQL_ConnString, 
	);
END_IF

END_PROGRAM

// Device/Application/MySQL_VISU
PROGRAM MySQL_VISU
VAR
	// ** MySQL_Connection String Handler FB - Do Not Edit INPUTs
	MySQL_ConnString		: MySQL.MySQL_ConnectionString;
		
	// ** MySQL_Open FB
	MySQL_Open				: MySQL.MySQL_Open;
	
	// ** Connection Parameters
	sHost					: STRING := 'localhost';			// Hostname or IP-adress
	uiPort					: UINT 	 := 3306;					// MySQL Server Port
	sDatabase				: STRING := 'testdb';				// Database Name
	sUsername				: STRING := 'root';					// Database Username
	sPassword				: STRING := 'root';					// User password 
	xDoOpen		 			: BOOL;								// Start opening the Connection
	
	// ** MySQL_Execute FB 
	MySQL_Exec: MySQL.MySQL_Exec;
	
	MySQL_Command_Exec		: ARRAY [0..gc_MySQL_iStatementMax] OF STRING(gc_MySQL_iStatementLength);// := ['INSERT INTO data (Column_1, Column_2, Column_3) VALUES (1, 5, 10)'];
	xDoExecute	 			: BOOL;								// Start Execute MySQL Exec

	// ** Dynamic Execute String
	iVar1					: INT := 1;
	iVar2					: INT := 2;
	iVar3					: INT := 3;
	
	// ** MySQL_Query FB
	MySql_Query				: MySQL.MySql_Query;	
	MySQL_Command_Query		: ARRAY [0..gc_MySQL_iStatementMax] OF STRING(gc_MySQL_iStatementLength); // := ['SELECT * from data'];
	xDoQuery				: BOOL;								// Start 
	
	// ** MySQL_GetStringValue function
	iRow					: INT; 								// Row index
	iColumn					: INT;								// Column index
	
	stResult 				: MySQL.MySQL_DataSet; 				// Result Structure
	
	ReadableString			: STRING(500); 						// Readable String	
	
	// ** MySQL_Close FB
	MySQL_Close				: MySQL.MySQL_Close;
	xDoClose 				: BOOL;
END_VAR

END_PROGRAM

// Device/Application/Operator_panel
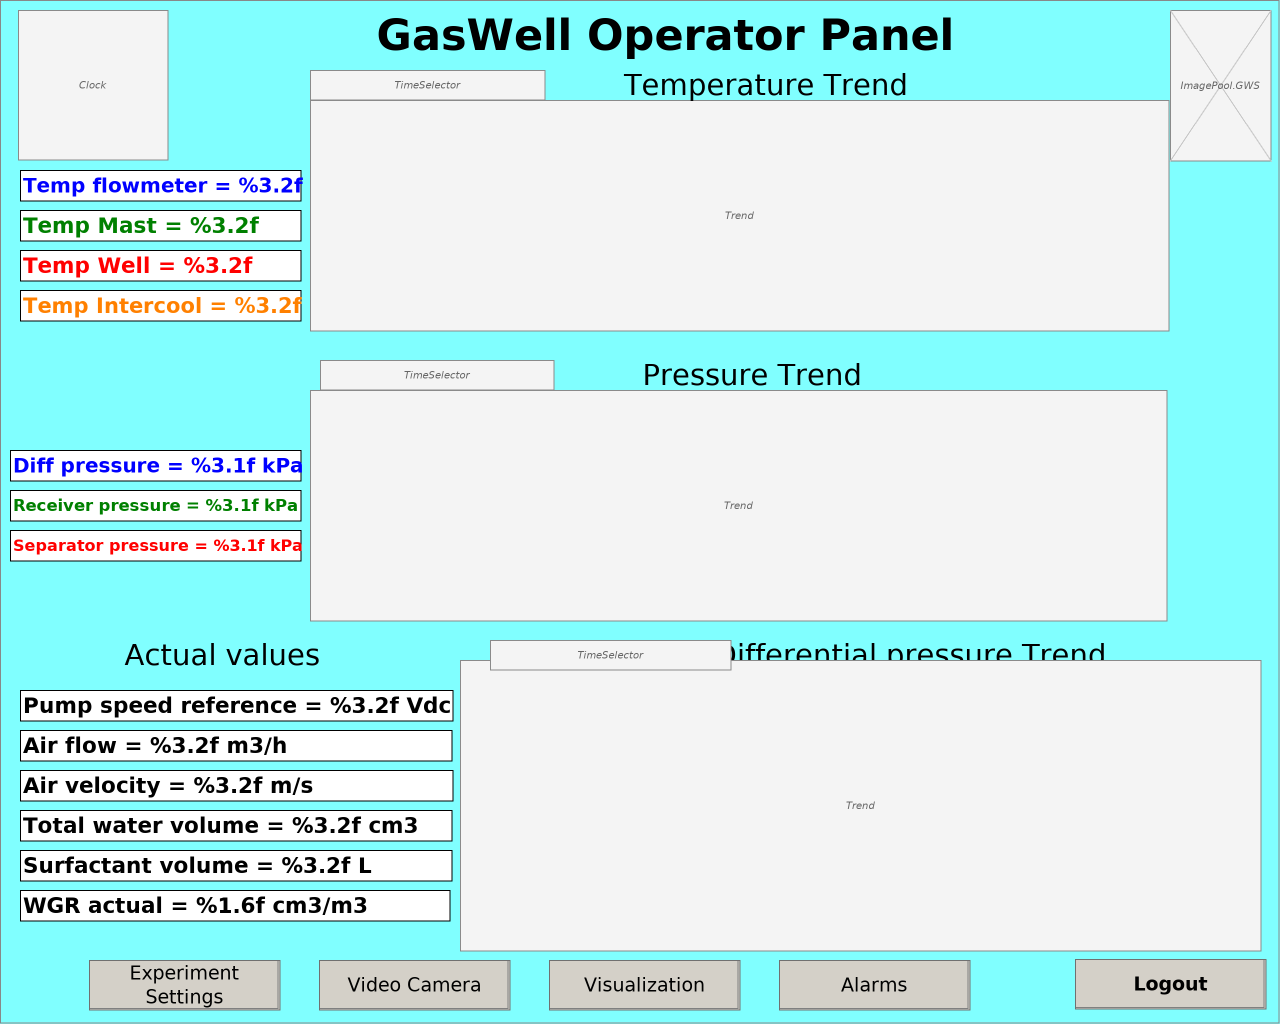
VISUALIZATION Operator_panel  // 1280x1024
    Label (360,10 611x50), "GasWell Operator Panel"
    Rectangle (20,170 281x31), "Temp flowmeter = %3.2f", text variable: PLC_PRG.Air_temp
    Trend (310,100 859x231)
        p2423372160: HH:mm:ss
        p2833066001: Visualization_Trend2
        p2541140726: Trend1TimeSelector
    Image (1170,10 101x151), image: ImagePool.GWS
    Clock (18,10 150x150)
        p1016715431: Element-Clock-Green
    Rectangle (20,210 281x31), "Temp Mast = %3.2f", text variable: GVL.Mast_temperature
    Rectangle (20,250 281x31), "Temp Well = %3.2f", text variable: GVL.Well_temperature
    Label (640,70 252x30), "Temperature Trend"
    Trend (310,390 857x231)
        p2423372160: HH:mm:ss
        p2833066001: Visualization_Trend3
        p2541140726: Trend2TimeSelector
    Label (640,360 225x30), "Pressure Trend"
    Rectangle (10,450 291x31), "Diff pressure = %3.1f kPa", text variable: PLC_PRG.Differential_pressure
    Rectangle (10,490 291x31), "Receiver pressure = %3.1f kPa", text variable: PLC_PRG.Receiver_pressure
    Rectangle (10,530 291x31), "Separator pressure = %3.1f kPa", text variable: PLC_PRG.Separator_pressure
    Button (89,960 191x50), "Experiment Settings"
        OnMouseClick:  Assign=Experiment_settings, Type=Assignment
    Button (319,960 191x50), "Video Camera"
    Button (549,960 191x50), "Visualization"
        OnMouseClick:  Assign=Visualization, Type=Assignment
    Rectangle (20,690 433x31), "Pump speed reference = %3.2f Vdc", text variable: PLC_PRG.OP_Speed_Pump
    Rectangle (20,730 432x31), "Air flow = %3.2f m3/h", text variable: PLC_PRG.Air_flow
    Rectangle (20,770 433x31), "Air velocity = %3.2f m/s", text variable: PLC_PRG.Air_velocity
    Rectangle (20,810 432x31), "Total water volume = %3.2f cm3", text variable: PLC_PRG.Waterflow_in
    Rectangle (20,850 432x31), "Surfactant volume = %3.2f L", text variable: PLC_PRG.Foam_volume_counts
    Label (110,640 225x30), "Actual values"
    Label (720,640 381x30), "Differential pressure Trend"
    Rectangle (20,890 430x31), "WGR actual = %1.6f cm3/m3", text variable: PLC_PRG.OP_WGR_Setpoint
    Button (779,960 191x50), "Alarms"
    Button (1075,959 191x50), "Logout"
        OnMouseDown:  Type=Logout
        OnMouseDown: execute {
            IF VisuElems.CurrentUserGroupId <> 0 THEN
            	VisuElems.g_VisuManager.SetMainVisu(pClientData, 'Login');
            END_IF
        }
    TimeSelector (310,70 235x30)
        p3737533738: GenElemInst_9
        p677259794: Zoom:
    TimeSelector (320,360 234x30)
        p3737533738: GenElemInst_34
        p677259794: Zoom:
    Trend (460,660 801x291)
        p758368661: dd-MMM-yy
        p2423372160: H:mm:ss:ms
        p2833066001: Operator_panel_Trend3
        p2541140726: Trend3TimeSelector
    TimeSelector (490,640 241x30)
        p3737533738: GenElemInst_103
        p677259794: Zoom:
    Rectangle (20,290 281x31), "Temp Intercool = %3.2f", text variable: PLC_PRG.Intercoller_temperature
END_VISUALIZATION

// Device/Application/Experiment_settings
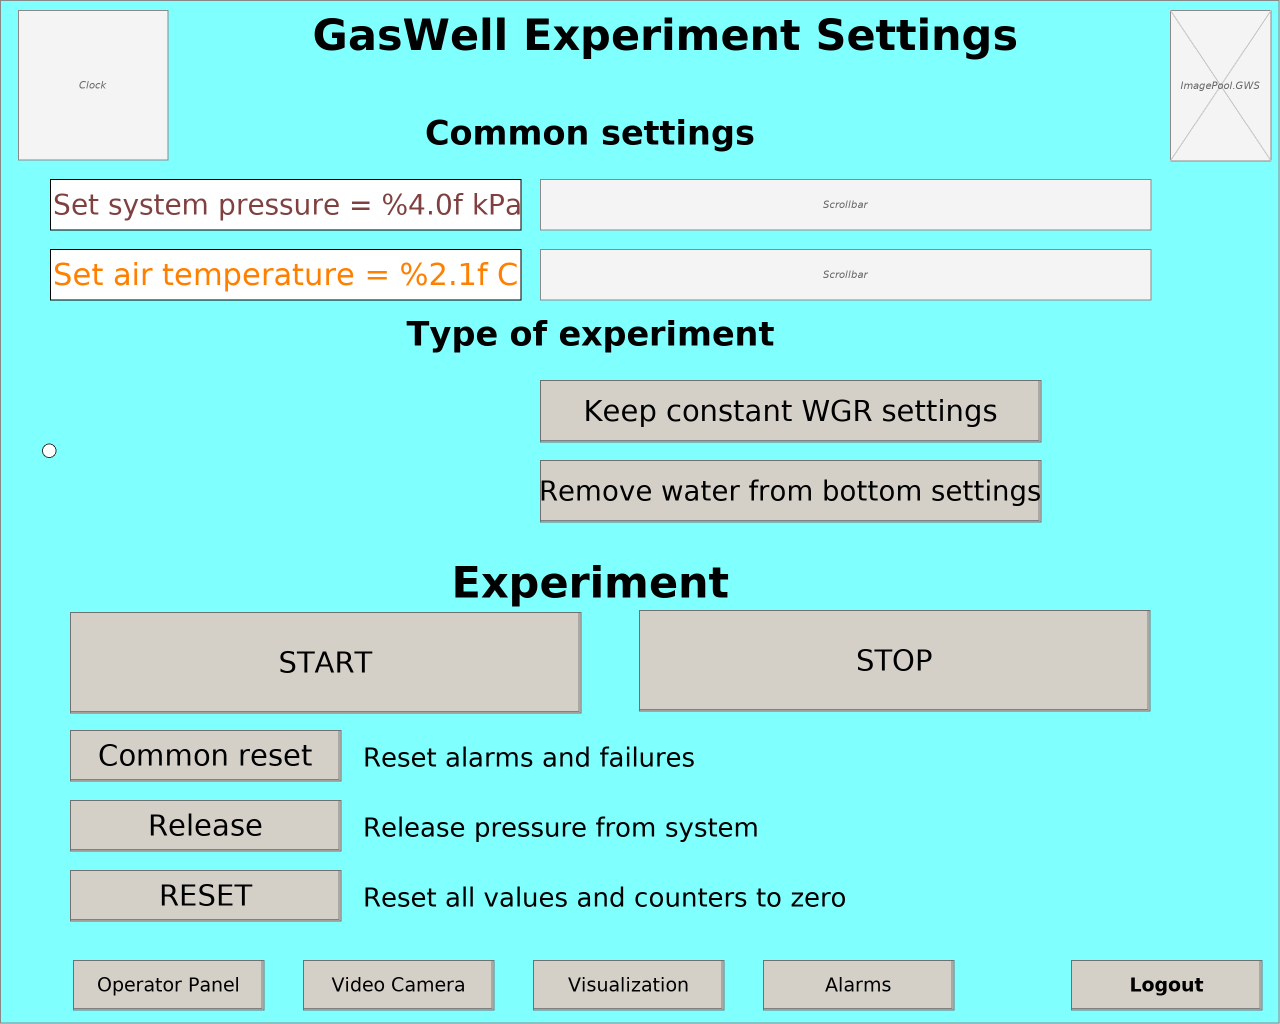
VISUALIZATION Experiment_settings  // 1280x1024
    Label (360,10 611x50), "GasWell Experiment Settings"
    Image (1170,10 101x151), image: ImagePool.GWS
    Clock (18,10 150x150)
        p1016715431: Element-Clock-Green
    Button (73,960 191x50), "Operator Panel"
        OnMouseClick:  Assign=Operator_panel, Type=Assignment
    Button (303,960 191x50), "Video Camera"
    Button (533,960 191x50), "Visualization"
        OnMouseClick:  Assign=Visualization, Type=Assignment
    Rectangle (50,179 471x51), "Set system pressure = %4.0f kPa", text variable: PLC_PRG.OP_System_Pressure
        OnMouseClick: write the text variable via VisuDialogs.Numpad, min 0, max 1000
    Rectangle (50,249 471x51), "Set air temperature = %2.1f C", text variable: PLC_PRG.OP_System_Temperature
        OnMouseClick: write the text variable via VisuDialogs.Numpad, min 10, max 50
    Scrollbar (540,249 611x51)
        p1057716461: PLC_PRG.OP_System_Temperature
    Scrollbar (540,179 611x51)
        p1057716461: PLC_PRG.OP_System_Pressure
    Label (460,560 261x45), "Experiment"
    Button (70,612 511x101), "START"
        toggle PLC_PRG.START p2164770859=TRUE
        OnMouseDown:  ToggleVariable=PLC_PRG.START
    Button (639,610 511x101), "STOP"
        toggle PLC_PRG.STOP p2164770859=TRUE
        OnMouseDown:  ToggleVariable=PLC_PRG.STOP
    Button (70,730 271x51), "Common reset"
        toggle PLC_PRG.Common_RESET p2164770859=TRUE
        OnMouseDown:  ToggleVariable=PLC_PRG.Common_RESET
    Label (360,740 551x35), "Reset alarms and failures"
    Button (763,960 191x50), "Alarms"
    Button (1071,960 191x50), "Logout"
        OnMouseDown:  Type=Logout
        OnMouseDown: execute {
            IF VisuElems.CurrentUserGroupId <> 0 THEN
            	VisuElems.g_VisuManager.SetMainVisu(pClientData, 'Login');
            END_IF
        }
    Button (540,380 501x62), "Keep constant WGR settings"
        OnMouseClick:  Dialog=Settings_WGR, OpenModal=True, OpenCentered=True
    Label (430,311 321x45), "Type of experiment"
    Label (439,110 302x45), "Common settings"
    RadioButton (40,400 451x101), variable: PLC_PRG.Type_of_exp
        Areas[0]: Text=Keep constant WGR
        Areas[1]: Text=Remove water from the bottom
    Button (540,460 501x62), "Remove water from bottom settings"
    Button (70,800 271x51), "Release"
        toggle PLC_PRG.Release_pressure p2164770859=TRUE
        OnMouseDown:  ToggleVariable=PLC_PRG.Release_pressure
    Label (360,810 371x35), "Release pressure from system"
    Button (70,870 271x51), "RESET"
        toggle PLC_PRG.RESET_to_zero p2164770859=TRUE
        OnMouseDown:  ToggleVariable=PLC_PRG.RESET_to_zero
    Label (360,880 551x35), "Reset all values and counters to zero"
END_VISUALIZATION

// Device/Application/Login
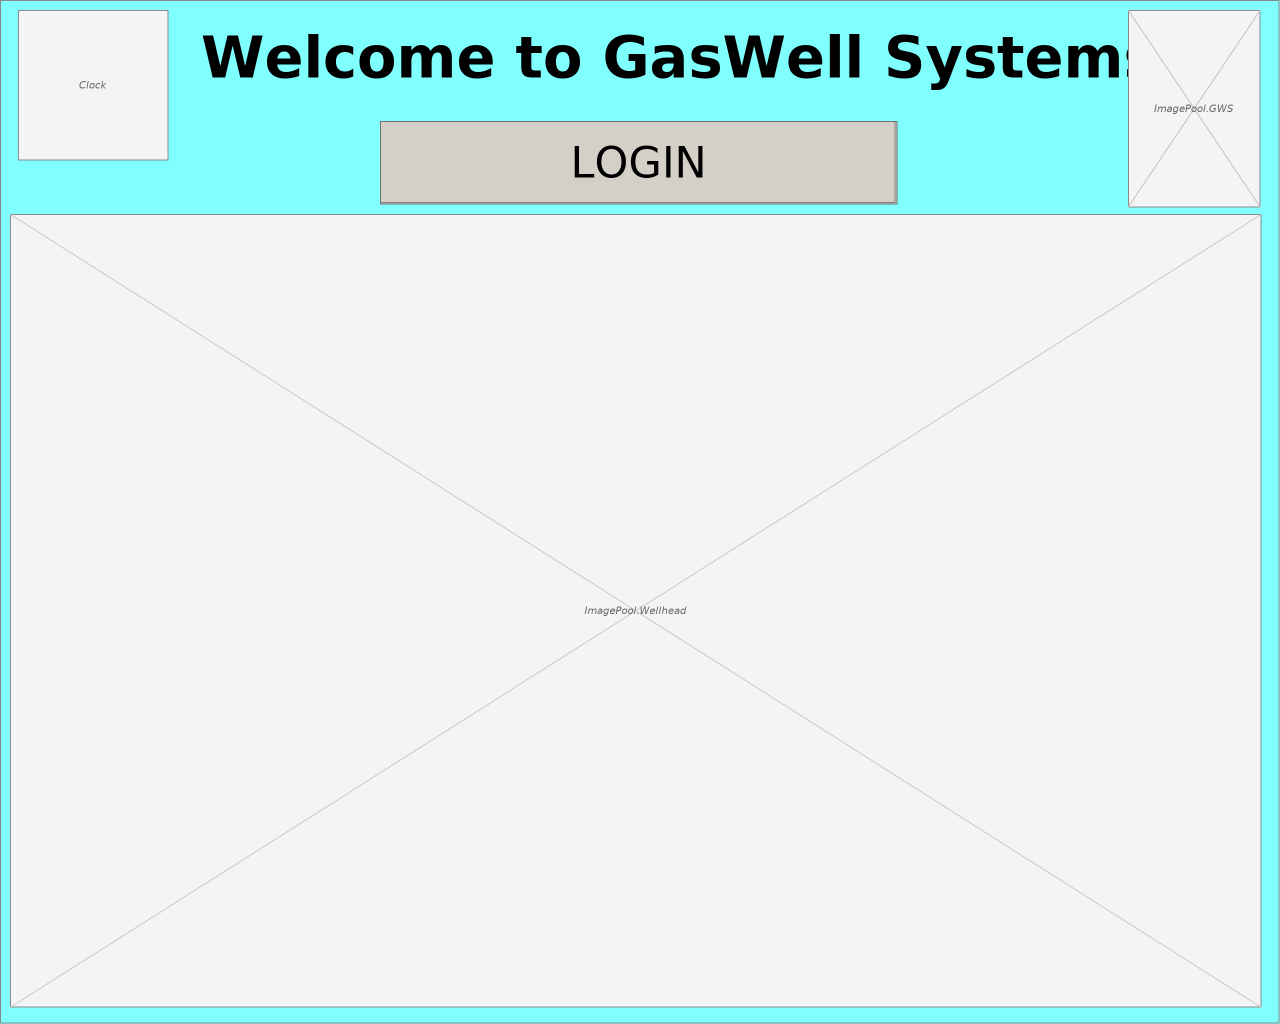
VISUALIZATION Login  // 1280x1024
    Label (211,18 937x78), "Welcome to GasWell Systems"
    Image (1128,10 132x197), image: ImagePool.GWS
    Clock (18,10 150x150)
        p1016715431: Element-Clock-Green
    Image (10,214 1251x793), image: ImagePool.Wellhead
    Button (380,121 517x83), "LOGIN"
        OnDialogClosed: execute { AfterLogin(pClientData); }
        OnMouseDown:  Type=Login
END_VISUALIZATION

// Device/Application/Settings_WGR
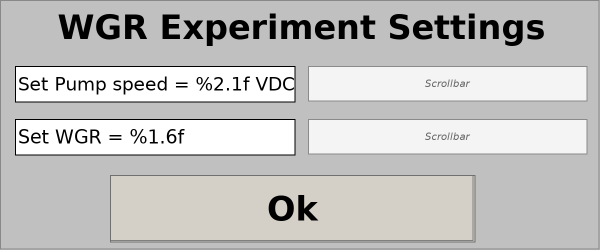
VISUALIZATION Settings_WGR  // 600x250
    Label (5,2 593x50), "WGR Experiment Settings"
    Button (110,175 365x67), "Ok"
        OnMouseClick:  Dialog=Settings_WGR, Result=OK, NumpadKeypadSet=True
    Scrollbar (308,66 279x35)
        p1057716461: PLC_PRG.OP_Speed_Pump
    Rectangle (15,66 280x36), "Set Pump speed = %2.1f VDC", text variable: PLC_PRG.OP_Speed_Pump
        OnMouseClick: write the text variable via VisuDialogs.Numpad, min 0, max 10
    Rectangle (15,119 280x36), "Set WGR = %1.6f", text variable: PLC_PRG.OP_WGR_Setpoint
        OnMouseClick: write the text variable via VisuDialogs.Numpad, min 0, max 0.01
    Scrollbar (308,119 279x35)
        p2245068023: 0.01
        p1057716461: PLC_PRG.OP_WGR_Setpoint
END_VISUALIZATION

// Device/Application/Visualization
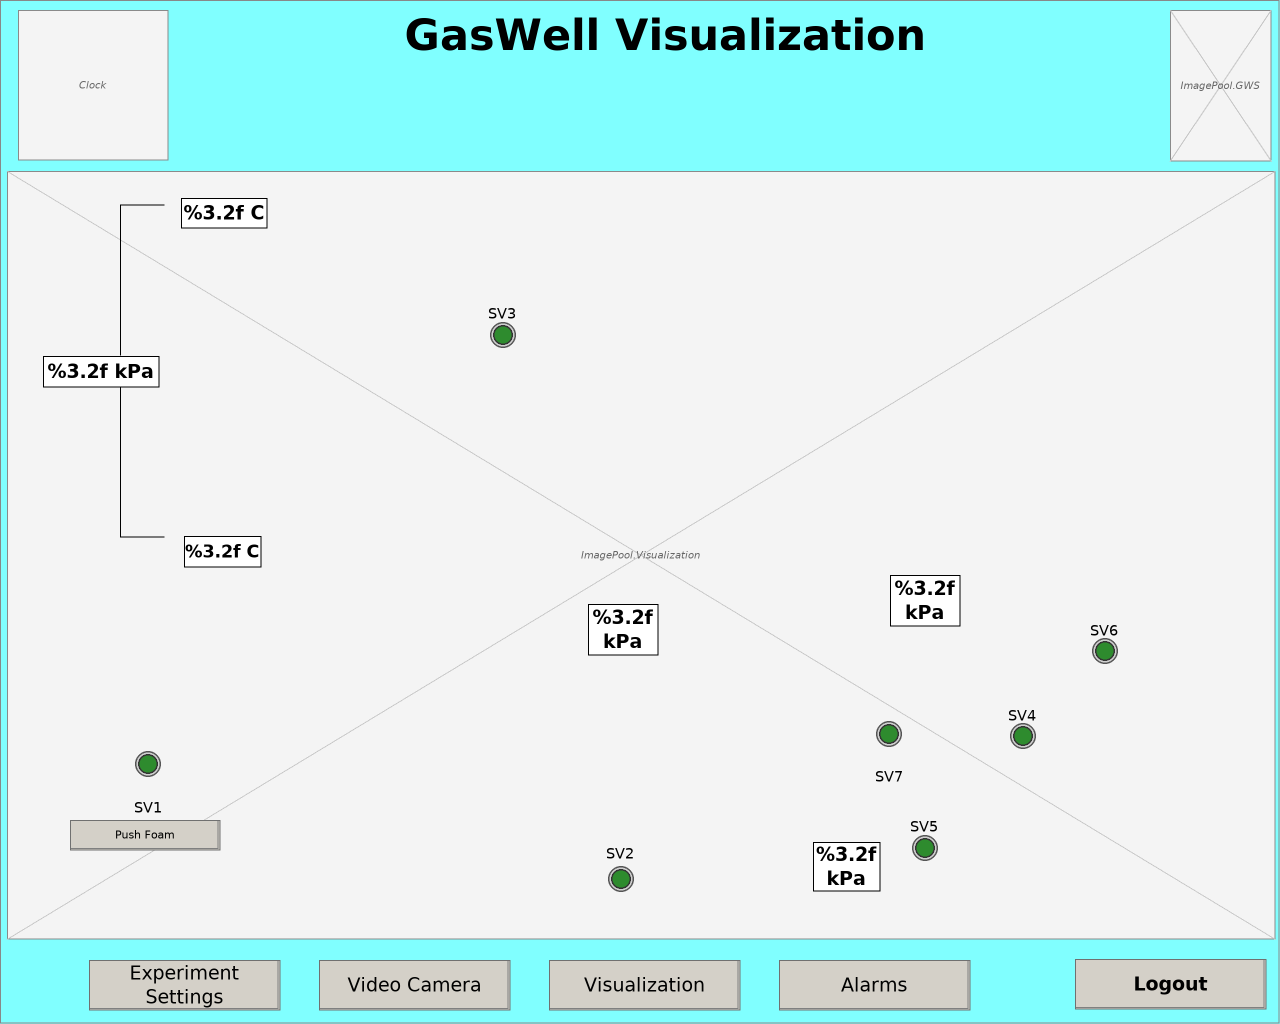
VISUALIZATION Visualization  // 1280x1024
    Image (7,171 1268x768), image: ImagePool.Visualization
    Label (360,10 611x50), "GasWell Visualization"
    Image (1170,10 101x151), image: ImagePool.GWS
    Clock (18,10 150x150)
        p1016715431: Element-Clock-Green
    Button (89,960 191x50), "Experiment Settings"
        OnMouseClick:  Assign=Experiment_settings, Type=Assignment
    Button (319,960 191x50), "Video Camera"
    Button (549,960 191x50), "Visualization"
    Button (779,960 191x50), "Alarms"
    Button (1075,959 191x50), "Logout"
        OnMouseDown:  Type=Logout
        OnMouseDown: execute {
            IF VisuElems.CurrentUserGroupId <> 0 THEN
            	VisuElems.g_VisuManager.SetMainVisu(pClientData, 'Login');
            END_IF
        }
    Rectangle (181,198 86x30), "%3.2f C", text variable: GVL.Mast_temperature
    Rectangle (184,536 77x31), "%3.2f C", text variable: GVL.Well_temperature
    Rectangle (43,356 116x31), "%3.2f kPa", text variable: PLC_PRG.Differential_pressure
    Line (120,205) (120,355)
    Line (164,205) (120,205)
    Line (120,387) (120,537)
    Line (164,537) (120,537)
    Rectangle (813,842 67x49), "%3.2f kPa", text variable: PLC_PRG.Receiver_pressure
    Rectangle (588,604 70x51), "%3.2f kPa", text variable: PLC_PRG.Separator_pressure
    Rectangle (890,575 70x51), "%3.2f kPa", text variable: PLC_PRG.Separator_pressure
    Lamp1 (133,749 30x30), variable: PLC_PRG.SV1_Switch_onoff, style: Lamp-Lamp1-Green
    Lamp1 (488,320 30x30), variable: PLC_PRG.SV3_Switch_onoff, style: Lamp-Lamp1-Green
    Lamp1 (606,864 30x30), variable: PLC_PRG.SV2_Switch_onoff, style: Lamp-Lamp1-Green
    Lamp1 (910,833 30x30), variable: PLC_PRG.SV5_Switch_onoff, style: Lamp-Lamp1-Green
    Lamp1 (874,719 30x30), variable: PLC_PRG.SV7_Switch_onoff, style: Lamp-Lamp1-Green
    Lamp1 (1008,721 30x30), variable: PLC_PRG.SV4_Switch_onoff, style: Lamp-Lamp1-Green
    Lamp1 (1090,636 30x30), variable: PLC_PRG.SV6_Switch_onoff, style: Lamp-Lamp1-Green
    Label (131,796 34x23), "SV1"
    Label (603,842 34x23), "SV2"
    Label (485,302 34x23), "SV3"
    Label (907,815 34x23), "SV5"
    Label (872,765 34x23), "SV7"
    Label (1005,704 34x23), "SV4"
    Label (1087,619 34x23), "SV6"
    Button (70,820 150x30), "Push Foam"
        OnMouseClick:  ToggleVariable=PLC_PRG.Push_foam
END_VISUALIZATION

// Device/Application/Well_not_killed_10min
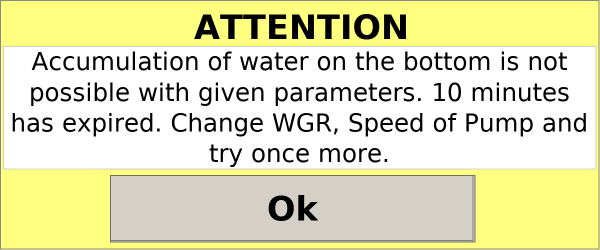
VISUALIZATION Well_not_killed_10min  // 600x250
    Label (5,2 593x50), "ATTENTION"
    Button (110,175 365x67), "Ok"
        OnMouseClick:  Dialog=Well_not_killed_10min, Result=OK, NumpadKeypadSet=True
    Textfield (3,46 593x123), "Accumulation of water on the bottom is not possible with given parameters. 10 minutes has expired. Change WGR, Speed of Pump and try once more."
END_VISUALIZATION

// Device/Application/MySQL_visu
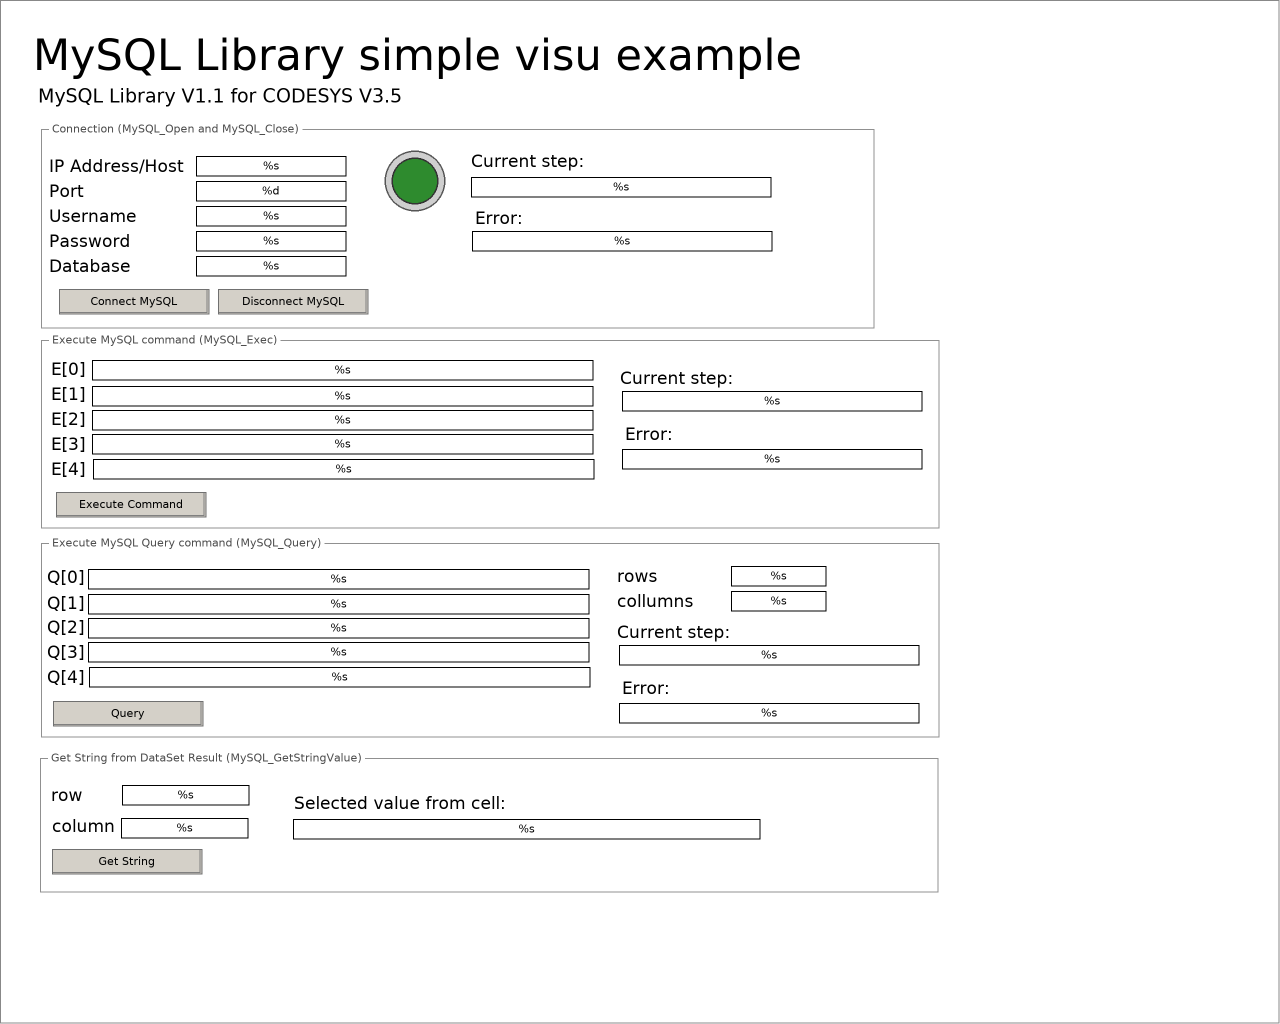
VISUALIZATION MySQL_visu  // 1280x1024
VAR_IN_OUT
	
END_VAR

VAR
	Execute0 : STRING;
	Execute1 : STRING;
	Execute2 : STRING;
	Execute3 : STRING;
	Execute4 : STRING;
	
	Q0 : STRING;
	Q1 : STRING;
	Q2 : STRING;
	Q3 : STRING;
	Q4 : STRING;
	
	row : INT;
	column : INT; 
END_VAR
    Label (35,80 508x32), "MySQL Library V1.1 for CODESYS V3.5"
    Label (30,30 957x50), "MySQL Library simple visu example"
    Label (46,156 150x20), "IP Address/Host"
    Label (46,181 150x20), "Port"
    Label (46,206 150x20), "Username"
    Label (46,231 150x20), "Password"
    Label (46,256 150x20), "Database"
    Rectangle (196,156 150x20), "%s", text variable: MySQL_VISU.sHost
        OnMouseClick: write the text variable via Default
    Rectangle (196,181 150x20), "%d", text variable: MySQL_VISU.uiPort
        OnMouseClick: write the text variable via Default
    Rectangle (196,206 150x20), "%s", text variable: MySQL_VISU.sUsername
        OnMouseClick: write the text variable via Default
    Rectangle (196,231 150x20), "%s", text variable: MySQL_VISU.sPassword
        OnMouseClick: write the text variable via Default, password
    Rectangle (196,256 150x20), "%s", text variable: MySQL_VISU.sDatabase
        OnMouseClick: write the text variable via Default
    Label (468,151 150x20), "Current step:"
    Label (472,208 150x20), "Error:"
    Rectangle (471,177 300x20), "%s", text variable: MySQL_VISU.MySQL_Open.sExeute_State
    Rectangle (472,231 300x20), "%s", text variable: MySQL_VISU.MySQL_Open.eError
    Button (59,289 150x25), "Connect MySQL"
        toggle MySQL_VISU.xDoOpen
    Button (218,289 150x25), "Disconnect MySQL"
        toggle MySQL_VISU.xDoClose
    Lamp1 (380,146 70x70), variable: MySQL_VISU.MySQL_Open.xConnected, style: Lamp-Lamp1-Green
    GroupBox (41,121 833x207), "Connection (MySQL_Open and MySQL_Close)"
    Button (56,492 150x25), "Execute Command"
        OnMouseDown: execute { MySQL_VISU.xDoExecute := FALSE; }
        OnMouseClick: execute {
            MySQL_VISU.MySQL_Command_Exec[0] := Execute0;
            MySQL_VISU.MySQL_Command_Exec[1] := Execute1;
            MySQL_VISU.MySQL_Command_Exec[2] := Execute2;
            MySQL_VISU.MySQL_Command_Exec[3] := Execute3;
            MySQL_VISU.MySQL_Command_Exec[4] := Execute4;
            MySQL_VISU.xDoExecute := TRUE;
        }
    Label (48,359 105x20), "E[0]"
    Label (48,384 105x20), "E[1]"
    Label (48,409 105x20), "E[2]"
    Label (48,434 105x20), "E[3]"
    Label (48,459 105x20), "E[4]"
    Rectangle (92,360 501x20), "%s", text variable: This^.Execute0
        OnMouseClick: write the text variable via Default
    Rectangle (92,386 501x20), "%s", text variable: This^.Execute1
        OnMouseClick: write the text variable via Default
    Rectangle (92,410 501x20), "%s", text variable: This^.Execute2
        OnMouseClick: write the text variable via Default
    Rectangle (92,434 501x20), "%s", text variable: This^.Execute3
        OnMouseClick: write the text variable via Default
    Rectangle (93,459 501x20), "%s", text variable: This^.Execute4
        OnMouseClick: write the text variable via Default
    Label (617,368 150x20), "Current step:"
    Rectangle (622,391 300x20), "%s", text variable: MySQL_VISU.MySQL_Exec.sExecute_State
    Rectangle (622,449 300x20), "%s", text variable: MySQL_VISU.MySQL_Exec.eError
    Label (622,424 150x20), "Error:"
    GroupBox (41,332 898x196), "Execute MySQL command (MySQL_Exec)"
    GroupBox (41,535 898x202), "Execute MySQL Query command (MySQL_Query)"
        Label (573,31 105x20), "rows"
        Rectangle (690,31 95x20), "%s", text variable: MySQL_VISU.stResult.uiRowCount
        Label (3,82 105x20), "Q[2]"
        Label (3,107 105x20), "Q[3]"
        Label (3,132 105x20), "Q[4]"
        Rectangle (47,59 501x20), "%s", text variable: This^.Q1
            OnMouseClick: write the text variable via Default
        Rectangle (47,83 501x20), "%s", text variable: This^.Q2
            OnMouseClick: write the text variable via Default
        Rectangle (47,107 501x20), "%s", text variable: This^.Q3
            OnMouseClick: write the text variable via Default
        Rectangle (48,132 501x20), "%s", text variable: This^.Q4
            OnMouseClick: write the text variable via Default
        Button (12,166 150x25), "Query"
            OnMouseDown: execute { MySQL_VISU.xDoQuery := FALSE; }
            OnMouseClick: execute {
                MySQL_VISU.MySQL_Command_Query[0] := Q0;
                MySQL_VISU.MySQL_Command_Query[1] := Q1;
                MySQL_VISU.MySQL_Command_Query[2] := Q2;
                MySQL_VISU.MySQL_Command_Query[3] := Q3;
                MySQL_VISU.MySQL_Command_Query[4] := Q4;
                MySQL_VISU.xDoQuery := TRUE;
            }
        Label (573,87 150x20), "Current step:"
        Rectangle (578,110 300x20), "%s", text variable: MySQL_VISU.MySql_Query.sExecute_State
        Rectangle (578,168 300x20), "%s", text variable: MySQL_VISU.MySql_Query.eError
        Label (578,143 150x20), "Error:"
        Label (3,32 105x20), "Q[0]"
        Label (3,58 105x20), "Q[1]"
        Rectangle (690,56 95x20), "%s", text variable: MySQL_VISU.stResult.uiColumnCount
        Label (573,56 105x20), "collumns"
        Rectangle (47,34 501x20), "%s", text variable: This^.Q0
            OnMouseClick: write the text variable via Default
    GroupBox (40,750 898x142), "Get String from DataSet Result (MySQL_GetStringValue)"
        Label (8,35 105x20), "row"
        Label (9,66 105x20), "column"
        Rectangle (253,69 467x20), "%s", text variable: MySQL_VISU.ReadableString
        Label (251,43 226x20), "Selected value from cell:"
        Rectangle (81,68 127x20), "%s", text variable: This^.column
            OnMouseClick: write the text variable via Default
        Rectangle (82,35 127x20), "%s", text variable: This^.row
            OnMouseClick: write the text variable via Default
    Button (52,849 150x25), "Get String"
        OnMouseClick: execute { MySQL_VISU.iRow := row; MySQL_VISU.iColumn := column; }
    Rectangle (40,895 900x15)
END_VISUALIZATION
